(* CODESYS project SPT_Kinematics.library
   Placeholder: SPT Kinematics
   Title: SPT Kinematics
   Version: 3.3.5
   Company: Beckhoff Automation LLC

Project tree, tasks and I/O mapping:
  libraries: SPT Base Types, * (Beckhoff Automation LLC); SPT Components, * (Beckhoff Automation LLC); SPT Event Logger, * (Beckhoff Automation LLC); Tc2_MC2, * (Beckhoff Automation GmbH); Tc2_MC2_Camming, * (Beckhoff Automation GmbH); Tc2_NcKinematicTransformation, * (Beckhoff Automation GmbH); Tc2_Standard, * (Beckhoff Automation GmbH); Tc2_System, * (Beckhoff Automation GmbH); Tc3_EventLogger, * (Beckhoff Automation GmbH); Tc3_McCoordinatedMotion, * (Beckhoff Automation GmbH)
  DUTs/
    KinematicComponentAmp/
      Enumerations/
        data type E_InitializeState_KinematicAmp
      HMI/
        data type ST_KinematicComponentAmp_Command
        data type ST_KinematicComponentAmp_Config
        data type ST_KinematicComponentAmp_HMI
        data type ST_KinematicComponentAmp_Status
      data type ST_AmpPoint
      data type ST_AmpPointCircular
      data type ST_KinematicComponentAmp_CmGroupState
    KinematicComponentBase/
      Enumerations/
        data type E_InitializeState_KinematicComponent
        data type E_KinematicDOF
        data type E_KinematicEnableSeq
      HMI/
        data type ST_KinematicComponent_Command
        data type ST_KinematicComponent_Config
        data type ST_KinematicComponent_HMI
        data type ST_KinematicComponent_Status
        data type ST_KinematicJogCommand
      data type ST_BasePoint
      data type ST_KinematicMotionParameter
      data type ST_KinematicMotionParameterValues
      data type ST_KinematicPosition
    KinematicComponentCamming/
      Enumerations/
        data type E_InitializeState_KinematicCamming
      HMI/
        data type ST_KinematicComponentCam_Command
        data type ST_KinematicComponentCam_Config
        data type ST_KinematicComponentCam_HMI
        data type ST_KinematicComponentCam_Status
      data type ST_CamTableSlaveDynamics
    KinematicGroup/
      HMI/
        data type ST_KinematicGroup_Command
        data type ST_KinematicGroup_Config
        data type ST_KinematicGroup_HMI
        data type ST_KinematicGroup_Status
      data type E_ChangeParameterSeq
      data type E_InitializeState_KinematicGroup
      data type E_KinematicPositionCalculationSeq
    data type E_AcsJoint
    data type E_McsAxis
  FunctionBlocks/
    function block FB_ComponentKinematicBase [ST]: CreateEvents, HMICommunication, Monitoring, Reset, CyclicLogic, ActPosition, Enabled, InPosition, Moving, Disable, Enable, JogCartesianAxis, JogJoint, Override, Stop, TargetMotionParameter, BuildKinGroup, DissolveKinGroup, KinematicEnableSeq, McResetAllAxis, iAxisRef, Initialize
    function block FB_ComponentKinematicMotionAmp [ST]: CreateEvents, HMICommunication, Monitoring, Reset, CyclicLogic, Moving, Override, Stop, CmIdentAxis1, CmIdentAxis2, CmIdentAxis3, CmIdentAxis4, ConveyorRef, BuildCmGroup, ClearPath, CmGroupRef, CmState, DisableCmGroup, EnableCmGroup, SetCoordinateTransform, StartMovePath, TrackConveyorBelt, UngroupCmGroup, AddCircularMoveToPath, AddLinearMoveToPath, MoveToPointCartesian, ChangeOccurred, GetPoint, Points, SetPoint, Initialize
    function block FB_ComponentKinematicMotionCamming [ST]: CreateEvents, HMICommunication, Monitoring, Reset, CyclicLogic, Disable, Enable, Override, Stop, CamClearPath, CamIn, CamMasterZero, CammingActive, CamOut, CamStartMovePath, BuildKinGroup, DissolveKinGroup, ReadCamTableSlaveDynamicsACS, ReadCamTableSlaveDynamicsMCS, CamAddMotionPointByAxis, CamAddPointToPath, ChangeOccurred, GetPoint, Points, SetPoint, CamInOptionsACS, CamInOptionsMCS, CamMasterAcs, CamMasterMcs, CamTableSlaveDynamicsACS, CamTableSlaveDynamicsMCS, Initialize
    function block FB_KinematicAxisRef [ST]: ACS, AcsAxisCount, AcsPositionAbsolute, DegreesOfFreedomConfigured, MCS
    function block FB_KinematicCamming [ST]: CyclicLogic, CamClearPath, CamIn, CamMasterZero, CammingActive, CamOut, CamStartMovePath, CamAddMotionPointByAxis, CamAddPointToPath, CamTableAddStartPoint, Disable, Enable, ReadCamTableSlaveDynamics, Reset, SetOverride, Stop, CamAxisCount, CamAxisRef, CamInOptions, CamMaster, CamTableSlaveDynamics, Initialize
    function block FB_KinematicGroup [ST]: CreateEvents, HMICommunication, Monitoring, Reset, CyclicLogic, ActivateExtRotationRange, BuildKinGroup, DeactivateExtRotationRange, DissolveKinGroup, PresetRotationExtRotationRange, ResetKinGroup, SetKinematicParameter, KinematicStatus, KinMetaInfo, OidKinTrafo, OidKinTrafoTool, CalcKinPosition, ChangeKinematicParameter, KinematicAxisIds, Initialize
    function block FB_KinematicMotionAmpBase [ST]: CyclicLogic, BuildCmGroup, ClearPath, DisableCmGroup, EnableCmGroup, SetCoordinateTransform, StartMovePath, TrackConveyorBelt, UngroupCmGroup, CmIdentAxis1, CmIdentAxis2, CmIdentAxis3, CmIdentAxis4, ConveyorRef, CmGroupRef, CmState, AddCircularMoveToPath, AddLinearMoveToPath, MapStatus, Reset, SetOverride, Stop, CmAxisCount, CmAxisRef, Initialize
    function block FB_RingBuffer_AmpAmpPath [ST]: ClearPath, CurrentFB, GetNewFb, Path
  GVLs/
    global variables KINEMATIC_CONSTANTS
  Interfaces/
    interface I_Kinematic: Disable, Enable, JogCartesianAxis, JogJoint, Stop, ActPosition, Enabled, InPosition, Moving, Override, TargetMotionParameter
    interface I_KinematicAxisRef: ACS, AcsAxisCount, AcsPositionAbsolute, DegreesOfFreedomConfigured, MCS
    interface I_KinematicCamming: CamClearPath, CamIn, CamMasterZero, CamOut, CamStartMovePath, CammingActive
    interface I_KinematicCm: BuildCmGroup, ClearPath, DisableCmGroup, EnableCmGroup, SetCoordinateTransform, StartMovePath, TrackConveyorBelt, UngroupCmGroup, CmIdentAxis1, CmIdentAxis2, CmIdentAxis3, CmIdentAxis4, ConveyorRef, CmGroupRef, CmState
    interface I_KinematicGroup: ActivateExtRotationRange, BuildKinGroup, DeactivateExtRotationRange, DissolveKinGroup, PresetRotationExtRotationRange, ResetKinGroup, SetKinematicParameter, KinematicStatus, KinMetaInfo, OidKinTrafo, OidKinTrafoTool
  Project Information/
    function F_GetCompany [ST]
    function F_GetTitle [ST]
    function F_GetVersion [ST]
  Utilities/
    function F_ADSErrorCodeExt [ST]
  Version/
    global variables Global_Version
  00000000-0000-0000-0000-000000000000|LICENSE
  LICENSE
  global variables Parameter_Kinematic
*)

// DUTs/KinematicComponentAmp/Enumerations/E_InitializeState_KinematicAmp
{attribute 'qualified_only'}
{attribute 'strict'}
TYPE E_InitializeState_KinematicAmp : (
		eInitializeState_Start := 0,
		eInitializeState_CheckLinking,
		eInitializeState_Done,
		eInitializeState_Failed
	);
END_TYPE

// DUTs/KinematicComponentAmp/HMI/ST_KinematicComponentAmp_Command
TYPE ST_KinematicComponentAmp_Command :
	STRUCT
		BuildCmGroup	: BOOL;
		EnableCmGroup	: BOOL;
		PointSelect		: UDINT;
		MoveToPointCm	: BOOL;
		TeachPoint		: BOOL;
		DisableCmGroup	: BOOL;
		DissolveCmGroup : BOOL;
	END_STRUCT
END_TYPE

// DUTs/KinematicComponentAmp/HMI/ST_KinematicComponentAmp_Config
TYPE ST_KinematicComponentAmp_Config :
	STRUCT
		CustomOverride : BOOL := FALSE;
		CustomCommand  : DINT;
	END_STRUCT
END_TYPE

// DUTs/KinematicComponentAmp/HMI/ST_KinematicComponentAmp_HMI
TYPE ST_KinematicComponentAmp_HMI :
	STRUCT
		Config	: ST_KinematicComponentAmp_Config;
		Command : ST_KinematicComponentAmp_Command;
		Status	: ST_KinematicComponentAmp_Status;
	END_STRUCT
END_TYPE

// DUTs/KinematicComponentAmp/HMI/ST_KinematicComponentAmp_Status
TYPE ST_KinematicComponentAmp_Status :
	STRUCT
		CmState		  : ST_KinematicComponentAmp_CmGroupState;
		SelectedPoint : ST_AmpPoint;
	END_STRUCT
END_TYPE

// DUTs/KinematicComponentAmp/ST_AmpPoint
TYPE ST_AmpPoint EXTENDS ST_BasePoint :
	STRUCT
		CircularMove			 : ST_AmpPointCircular;
		Velocity				 : MC_LREAL			  := MC_INVALID;
		Acceleration			 : MC_LREAL			  := MC_DEFAULT;
		Deceleration			 : MC_LREAL			  := MC_DEFAULT;
		Jerk					 : MC_LREAL			  := MC_DEFAULT;
		BufferMode				 : MC_BUFFER_MODE	  := MC_BUFFER_MODE.mcAborting;
		TransitionMode			 : MC_TRANSITION_MODE := mcTransModeNone;
		TransitionParameter		 : ARRAY[1..2] OF LREAL;
		TransitionParameterCount : UDINT;
		InvokeId				 : UDINT;
	END_STRUCT
END_TYPE

// DUTs/KinematicComponentAmp/ST_AmpPointCircular
TYPE ST_AmpPointCircular :
	STRUCT
		IsCircularMove : BOOL;
		CircMode	   : MC_CIRC_MODE;
		AuxPoint	   : ARRAY[1..3] OF MC_LREAL;
		PathChoice	   : MC_CIRC_PATHCHOICE;
	END_STRUCT
END_TYPE

// DUTs/KinematicComponentAmp/ST_KinematicComponentAmp_CmGroupState
TYPE ST_KinematicComponentAmp_CmGroupState :
	STRUCT
		McToPlcCm					: CDT_MCTOPLC_GROUP_CM;
		GroupBuilt					: BOOL;
		GroupMoving					: BOOL;
		GroupHoming					: BOOL;
		GroupErrorStop				: BOOL;
		GroupNotReady				: BOOL;
		GroupStandby				: BOOL;
		GroupStopping				: BOOL;
		GroupDisabled				: BOOL;
		GroupTrackingInSync			: BOOL;
		GroupTrackingActive			: BOOL;
		GroupTrackingCommandAborted : BOOL;
		AllAxesStanding				: BOOL;
		ConstantVelocity			: BOOL;
		Accelerating				: BOOL;
		Decelerating				: BOOL;
		InPosition					: BOOL;
		Error						: BOOL;
		ErrorId						: UDINT;
	END_STRUCT
END_TYPE

// DUTs/KinematicComponentBase/Enumerations/E_InitializeState_KinematicComponent
{attribute 'qualified_only'}
{attribute 'strict'}
TYPE E_InitializeState_KinematicComponent : (
		eInitializeState_Start := 0,
		eInitializeState_CheckIft,
		eInitializeState_CheckAxisLinks,
		eInitializeState_SetAxisIds,
		eInitializeState_InitGroup,
		eInitializeState_Done
	);
END_TYPE

// DUTs/KinematicComponentBase/Enumerations/E_KinematicDOF
{attribute 'qualified_only'}
{attribute 'strict'}
TYPE E_KinematicDOF : (
		eKinematicDOF_2	  := 2, //
		eKinematicDOF_3	  := 3, //
		eKinematicDOF_4	  := 4, // 
		eKinematicDOF_5	  := 5, // 
		eKinematicDOF_6	  := 6, //
		eKinematicDOF_Max := 7	// 
	);
END_TYPE

// DUTs/KinematicComponentBase/Enumerations/E_KinematicEnableSeq
{attribute 'qualified_only'}
{attribute 'strict'}
TYPE E_KinematicEnableSeq : (
		eKinematicEnableSeq_Idle := 0,
		eKinematicEnableSeq_Start,
		eKinematicEnableSeq_ResetGroup,
		eKinematicEnableSeq_Enable,
		eKinematicEnableSeq_BuildGroup,
		eKinematicEnableSeq_Done
	);
END_TYPE

// DUTs/KinematicComponentBase/HMI/ST_KinematicComponent_Command
TYPE ST_KinematicComponent_Command :
	STRUCT
		Enable	: BOOL;
		Disable : BOOL;
		Stop	: BOOL;
		JogAxis : ARRAY[1..6] OF ST_KinematicJogCommand;
	END_STRUCT
END_TYPE

// DUTs/KinematicComponentBase/HMI/ST_KinematicComponent_Config
TYPE ST_KinematicComponent_Config :
	STRUCT
		KinematicType : E_KinematicDOF;
		AcsAxisCount  : UDINT;
	END_STRUCT
END_TYPE

// DUTs/KinematicComponentBase/HMI/ST_KinematicComponent_HMI
TYPE ST_KinematicComponent_HMI :
	STRUCT
		Config	: ST_KinematicComponent_Config;
		Command : ST_KinematicComponent_Command;
		Status	: ST_KinematicComponent_Status;
	END_STRUCT
END_TYPE

// DUTs/KinematicComponentBase/HMI/ST_KinematicComponent_Status
TYPE ST_KinematicComponent_Status :
	STRUCT
		Enabled		: BOOL;
		InPosition	: BOOL;
		Moving		: BOOL;
		ActPosition : ST_KinematicPosition;
	END_STRUCT
END_TYPE

// DUTs/KinematicComponentBase/HMI/ST_KinematicJogCommand
TYPE ST_KinematicJogCommand :
	STRUCT
		JogFast_Forward	 : BOOL;
		JogFast_Backward : BOOL;
		JogSlow_Forward	 : BOOL;
		JogSlow_Backward : BOOL;
	END_STRUCT
END_TYPE

// DUTs/KinematicComponentBase/ST_BasePoint
TYPE ST_BasePoint :
	STRUCT
		AcsPosition : ARRAY[1..KINEMATIC_CONSTANTS.DEGREES_OF_FREEDOM_MAX] OF LREAL;
		McsPosition : ARRAY[1..KINEMATIC_CONSTANTS.DEGREES_OF_FREEDOM_MAX] OF LREAL;
	END_STRUCT
END_TYPE

// DUTs/KinematicComponentBase/ST_KinematicMotionParameter
TYPE ST_KinematicMotionParameter :
	STRUCT
		Acs : ARRAY[1..KINEMATIC_CONSTANTS.DEGREES_OF_FREEDOM_MAX] OF ST_KinematicMotionParameterValues;
		Mcs : ARRAY[1..KINEMATIC_CONSTANTS.DEGREES_OF_FREEDOM_MAX] OF ST_KinematicMotionParameterValues;
	END_STRUCT
END_TYPE

// DUTs/KinematicComponentBase/ST_KinematicMotionParameterValues
TYPE ST_KinematicMotionParameterValues :
	STRUCT
		Position	 : LREAL;
		Acceleration : LREAL;
		Deceleration : LREAL;
		Jerk		 : LREAL;
	END_STRUCT
END_TYPE

// DUTs/KinematicComponentBase/ST_KinematicPosition
TYPE ST_KinematicPosition :
	STRUCT
		ACS : ARRAY[1..8] OF LREAL;
		MCS : ARRAY[1..8] OF LREAL;
	END_STRUCT
END_TYPE

// DUTs/KinematicComponentCamming/Enumerations/E_InitializeState_KinematicCamming
{attribute 'qualified_only'}
{attribute 'strict'}
TYPE E_InitializeState_KinematicCamming : (
		eInitializeState_Start := 0,
		eInitializeState_CheckLinking,
		eInitializeState_CheckRef,
		eInitializeState_Done,
		eInitializeState_Failed
	);
END_TYPE

// DUTs/KinematicComponentCamming/HMI/ST_KinematicComponentCam_Command
TYPE ST_KinematicComponentCam_Command :
	STRUCT
		CamAddPoint	   : BOOL;
		CamIn		   : BOOL;
		CamOut		   : BOOL;
		CamDeletePoint : BOOL;
		PointSelect	   : UDINT;
		MoveToPointCam : BOOL;
		TeachPoint	   : BOOL;
	END_STRUCT
END_TYPE

// DUTs/KinematicComponentCamming/HMI/ST_KinematicComponentCam_Config
TYPE ST_KinematicComponentCam_Config :
	STRUCT
		CustomOverride : BOOL := FALSE;
		CustomCommand  : DINT;
	END_STRUCT
END_TYPE

// DUTs/KinematicComponentCamming/HMI/ST_KinematicComponentCam_HMI
TYPE ST_KinematicComponentCam_HMI :
	STRUCT
		Config	: ST_KinematicComponentCam_Config;
		Command : ST_KinematicComponentCam_Command;
		Status	: ST_KinematicComponentCam_Status;
	END_STRUCT
END_TYPE

// DUTs/KinematicComponentCamming/HMI/ST_KinematicComponentCam_Status
TYPE ST_KinematicComponentCam_Status :
	STRUCT
		CammingActive : BOOL;
		SelectedPoint : ST_BasePoint;
	END_STRUCT
END_TYPE

// DUTs/KinematicComponentCamming/ST_CamTableSlaveDynamics
TYPE ST_CamTableSlaveDynamics :
	STRUCT
		SlavePosition	  : LREAL;
		SlaveVelocity	  : LREAL;
		SlaveAcceleration : LREAL;
	END_STRUCT
END_TYPE

// DUTs/KinematicGroup/HMI/ST_KinematicGroup_Command
TYPE ST_KinematicGroup_Command :
	STRUCT
		BuildGroup	  : BOOL;
		DissolveGroup : BOOL;
	END_STRUCT
END_TYPE

// DUTs/KinematicGroup/HMI/ST_KinematicGroup_Config
TYPE ST_KinematicGroup_Config :
	STRUCT
	END_STRUCT
END_TYPE

// DUTs/KinematicGroup/HMI/ST_KinematicGroup_HMI
TYPE ST_KinematicGroup_HMI :
	STRUCT
		Config	: ST_KinematicGroup_Config;
		Command : ST_KinematicGroup_Command;
		Status	: ST_KinematicGroup_Status;
	END_STRUCT
END_TYPE

// DUTs/KinematicGroup/HMI/ST_KinematicGroup_Status
TYPE ST_KinematicGroup_Status :
	STRUCT
		KinStatusReady : BOOL;
		KinStatus	   : E_KinStatus;
	END_STRUCT
END_TYPE

// DUTs/KinematicGroup/E_ChangeParameterSeq
{attribute 'qualified_only'}
{attribute 'strict'}
TYPE E_ChangeParameterSeq : (
		eChangeParameterSeq_Idle := 0,
		eChangeParameterSeq_Start,
		eChangeParameterSeq_Unlock,
		eChangeParameterSeq_Change,
		eChangeParameterSeq_ChangeDone,
		eChangeParameterSeq_Lock,
		eChangeParameterSeq_Error
	);
END_TYPE

// DUTs/KinematicGroup/E_InitializeState_KinematicGroup
{attribute 'qualified_only'}
{attribute 'strict'}
TYPE E_InitializeState_KinematicGroup : (
		eInitializeState_Start := 0,
		eInitializeState_CheckAxisIds,
		eInitializeState_CheckLinking,
		eInitializeState_CheckOid,
		eInitializeState_Done
	);
END_TYPE

// DUTs/KinematicGroup/E_KinematicPositionCalculationSeq
{attribute 'qualified_only'}
{attribute 'strict'}
TYPE E_KinematicPositionCalculationSeq : (
		eKinematicPositionCalculationSeq_Start := 0,
		eKinematicPositionCalculationSeq_Calc,
		eKinematicPositionCalculationSeq_Done
	);
END_TYPE

// DUTs/E_AcsJoint
{attribute 'qualified_only'}
TYPE E_AcsJoint : (
		Joint_1 := 1,
		Joint_2 := 2,
		Joint_3 := 3,
		Joint_4 := 4,
		Joint_5 := 5,
		Joint_6 := 6
	);
END_TYPE

// DUTs/E_McsAxis
{attribute 'qualified_only'}
TYPE E_McsAxis : (
		X	 := 1,
		Y	 := 2,
		Z	 := 3,
		Rot1 := 4, // C1, Rx,..
		Rot2 := 5, // C2, Ry,..
		Rot3 := 6  // C3, Rz,..
	);
END_TYPE

// GVLs/KINEMATIC_CONSTANTS
{attribute 'qualified_only'}
VAR_GLOBAL CONSTANT
	DEGREES_OF_FREEDOM_MAX : UINT := (TO_UINT(E_KinematicDOF.eKinematicDOF_Max) - 1);
END_VAR

// Version/Global_Version
{attribute 'TcGenerated'}
{attribute 'no-analysis'}
{attribute 'linkalways'}
// This function has been automatically generated from the project information.
VAR_GLOBAL CONSTANT
	{attribute 'const_non_replaced'}
	stLibVersion_SPT_Kinematics : ST_LibVersion := (iMajor := 3, iMinor := 3, iBuild := 5, iRevision := 0, nFlags := 1, sVersion := '3.3.5');
END_VAR

// Parameter_Kinematic
{attribute 'qualified_only'}
VAR_GLOBAL CONSTANT
	PathBufferSize				   : UDINT(4096..32768) := 4096;
	MaxPoints					   : UDINT(0..500)		:= 10;
	DefaultStopDeceleration		   : LREAL				:= 1000;  // mm/s^2 or deg/s^2
	DefaultStopDecelerationJerk	   : LREAL				:= 10000; // mm/s^3 or deg/s^3
	MaxCammingPositionsPerTable	   : UDINT(2..30)		:= 5;	  // Max Positions per move Command in Camming
	CamDefaultMoveVelocity		   : LREAL				:= 100;	  // mm/s or deg/s
	CamDefaultMoveAcceleration	   : LREAL				:= 1000;  // mm/s^2 or deg/s^2
	CamDefaultMoveDeceleration	   : LREAL				:= 1000;  // mm/s^2 or deg/s^2
	CamDefaultMoveJerk			   : LREAL				:= 10000; // mm/s^3 or deg/s^3		
	ExecuteCamPeriodically		   : BOOL				:= FALSE;
	CamMasterAbsolute			   : BOOL				:= TRUE;
	CamSlaveAbsolute			   : BOOL				:= TRUE;
	CammingFirstPointInTableByUser : BOOL				:= FALSE;
END_VAR

// FunctionBlocks/FB_ComponentKinematicBase
FUNCTION_BLOCK FB_ComponentKinematicBase EXTENDS FB_KinematicGroup IMPLEMENTS I_Kinematic
VAR
	// Kinematic Axis
	iAxis	 : I_KinematicAxisRef;
	_AxisAcs : REFERENCE TO ARRAY[1..KINEMATIC_CONSTANTS.DEGREES_OF_FREEDOM_MAX] OF AXIS_REF;
	_AxisMcs : REFERENCE TO ARRAY[1..KINEMATIC_CONSTANTS.DEGREES_OF_FREEDOM_MAX] OF AXIS_REF;

	// Internal Variables
	_KinematicComponentInit		: E_InitializeState_KinematicComponent;
	_KinematicEnableSeq			: E_KinematicEnableSeq := E_KinematicEnableSeq.eKinematicEnableSeq_Idle;
	_KinematicComponentBaseBusy : BOOL;
	_i							: UDINT;
	_ActPosition				: ST_KinematicPosition;
	_AcsSpeedOverride			: LREAL := 100.0;
	_McsSpeedOverride			: LREAL := 100.0;
	_McPowerAcsErrorActive		: BOOL;
	_McPowerMcsErrorActive		: BOOL;
	_TargetMotionParameter		: ST_KinematicMotionParameter;

	// MC Functions
	_McPowerACS : ARRAY[1..KINEMATIC_CONSTANTS.DEGREES_OF_FREEDOM_MAX] OF MC_POWER;
	_McPowerMCS : ARRAY[1..KINEMATIC_CONSTANTS.DEGREES_OF_FREEDOM_MAX] OF MC_POWER;
	_McJogACS	: ARRAY[1..KINEMATIC_CONSTANTS.DEGREES_OF_FREEDOM_MAX] OF MC_JOG;
	_McJogMCS	: ARRAY[1..KINEMATIC_CONSTANTS.DEGREES_OF_FREEDOM_MAX] OF MC_JOG;
	_McResetACS : ARRAY[1..KINEMATIC_CONSTANTS.DEGREES_OF_FREEDOM_MAX] OF MC_Reset;
	_McResetMCS : ARRAY[1..KINEMATIC_CONSTANTS.DEGREES_OF_FREEDOM_MAX] OF MC_Reset;
	_McHaltACS	: ARRAY[1..KINEMATIC_CONSTANTS.DEGREES_OF_FREEDOM_MAX] OF MC_Halt;
	_McHaltMCS	: ARRAY[1..KINEMATIC_CONSTANTS.DEGREES_OF_FREEDOM_MAX] OF MC_Halt;

	// HMI
	KinematicComponent_HMI : ST_KinematicComponent_HMI;

	// Alarms
	KinematicComponentBaseAlarms : ARRAY[1..KINEMATIC_COMPONENT_BASE_ALARM_COUNT] OF FB_TcAlarm;
END_VAR

VAR CONSTANT
	KINEMATIC_COMPONENT_BASE_ALARM_COUNT : UINT := 9;
END_VAR

//! @summary Initializes event function blocks using this components's name
{attribute 'call_after_online_change_slot' := '<slot>'}
METHOD PROTECTED CreateEvents

//! @description This method is called by <c>Initialize()</c> as required
F_CreateAllEventsInClass(Alarms		:= KinematicComponentBaseAlarms,
						 ClassSize	:= SIZEOF(TC_EVENTS.KinematicComponentBase),
						 pInitEvent := ADR(TC_EVENTS.KinematicComponentBase.InitReferenceEvent),
						 Prefix		:= Name);

SUPER^.CreateEvents();
END_METHOD

//! @summary Provides interlocks for HMI control and updates HMI status information for this component
METHOD PROTECTED HMICommunication

//! @description This method is called cyclically by <c>CyclicLogic()</c>
//Extend this method in extended FBs to communicate specific implementation data
SUPER^.HMICommunication();

// Kinematic HMI-Control
IF ComponentBase_HMI.Status.HMIControlAvailable THEN
	IF KinematicComponent_HMI.Command.Enable THEN
		THIS^.Enable();
		KinematicComponent_HMI.Command.Enable := FALSE;
	END_IF

	IF KinematicComponent_HMI.Command.Disable THEN
		THIS^.Disable();
		KinematicComponent_HMI.Command.Disable := FALSE;
	END_IF

	IF KinematicComponent_HMI.Command.Stop THEN
		Stop(0, 0);
		KinematicComponent_HMI.Command.Stop := FALSE;
	END_IF

	(*Jog*)
	FOR _i := 1 TO TO_UDINT(iAxis.DegreesOfFreedomConfigured) DO
		// Reset for Jogging-Function at HMI-control available
		THIS^.JogCartesianAxis(Axisx	:= _i,
							   Forward	:= FALSE,
							   Backward := FALSE,
							   JogMode	:= E_JogMode.MC_JOGMODE_STANDARD_SLOW);

		// Axis Jog Command
		IF SUPER^.KinematicStatus = E_KinStatus.KinStatus_Ready THEN // MCS-Axis active with Kinematic Model
			IF KinematicComponent_HMI.Command.JogAxis[_i].JogSlow_Forward THEN
				THIS^.JogCartesianAxis(Axisx	:= _i,
									   Forward	:= TRUE,
									   Backward := FALSE,
									   JogMode	:= E_JogMode.MC_JOGMODE_STANDARD_SLOW);
			ELSIF KinematicComponent_HMI.Command.JogAxis[_i].JogFast_Forward THEN
				THIS^.JogCartesianAxis(Axisx	:= _i,
									   Forward	:= TRUE,
									   Backward := FALSE,
									   JogMode	:= E_JogMode.MC_JOGMODE_STANDARD_FAST);
			ELSIF KinematicComponent_HMI.Command.JogAxis[_i].JogSlow_Backward THEN
				THIS^.JogCartesianAxis(Axisx	:= _i,
									   Forward	:= FALSE,
									   Backward := TRUE,
									   JogMode	:= E_JogMode.MC_JOGMODE_STANDARD_SLOW);
			ELSIF KinematicComponent_HMI.Command.JogAxis[_i].JogFast_Backward THEN
				THIS^.JogCartesianAxis(Axisx	:= _i,
									   Forward	:= FALSE,
									   Backward := TRUE,
									   JogMode	:= E_JogMode.MC_JOGMODE_STANDARD_FAST);
			END_IF
		END_IF
	END_FOR

	FOR _i := 1 TO TO_UDINT(iAxis.AcsAxisCount) DO
		// Reset for Jogging-Function at HMI-control available
		THIS^.JogJoint(Jointx	:= _i,
					   Forward	:= FALSE,
					   Backward := FALSE,
					   JogMode	:= E_JogMode.MC_JOGMODE_STANDARD_SLOW);

		// Axis Jog Command
		IF SUPER^.KinematicStatus = E_KinStatus.KinStatus_Empty THEN // ACS-Axis active
			IF KinematicComponent_HMI.Command.JogAxis[_i].JogSlow_Forward THEN
				THIS^.JogJoint(Jointx	:= _i,
							   Forward	:= TRUE,
							   Backward := FALSE,
							   JogMode	:= E_JogMode.MC_JOGMODE_STANDARD_SLOW);
			ELSIF KinematicComponent_HMI.Command.JogAxis[_i].JogFast_Forward THEN
				THIS^.JogJoint(Jointx	:= _i,
							   Forward	:= TRUE,
							   Backward := FALSE,
							   JogMode	:= E_JogMode.MC_JOGMODE_STANDARD_FAST);
			ELSIF KinematicComponent_HMI.Command.JogAxis[_i].JogSlow_Backward THEN
				THIS^.JogJoint(Jointx	:= _i,
							   Forward	:= FALSE,
							   Backward := TRUE,
							   JogMode	:= E_JogMode.MC_JOGMODE_STANDARD_SLOW);
			ELSIF KinematicComponent_HMI.Command.JogAxis[_i].JogFast_Backward THEN
				THIS^.JogJoint(Jointx	:= _i,
							   Forward	:= FALSE,
							   Backward := TRUE,
							   JogMode	:= E_JogMode.MC_JOGMODE_STANDARD_FAST);
			END_IF
		END_IF
	END_FOR
END_IF

// Status to HMI
KinematicComponent_HMI.Config.KinematicType := iAxis.DegreesOfFreedomConfigured;
KinematicComponent_HMI.Config.AcsAxisCount	:= iAxis.AcsAxisCount;
KinematicComponent_HMI.Status.Enabled		:= THIS^.Enabled;
KinematicComponent_HMI.Status.InPosition	:= THIS^.InPosition;
KinematicComponent_HMI.Status.Moving		:= THIS^.Moving;
KinematicComponent_HMI.Status.ActPosition	:= _ActPosition;
END_METHOD

//! Provides basic error detection and event handling for this component
METHOD PROTECTED Monitoring

(*! @descriptionThis method is called cyclically by <c>CyclicLogic()</c>*)
// Raise Error
SUPER^.Monitoring();
FOR _i := 1 TO TO_UDINT(iAxis.AcsAxisCount) DO
	IF _McPowerACS[_i].Error AND NOT KinematicComponentBaseAlarms[E_KinematicComponentBase.McPowerACS].bRaised THEN
		RaiseAlarmWithStrings(Alarm := KinematicComponentBaseAlarms[E_KinematicComponentBase.McPowerACS], F_ADSErrorCodeExt(_McPowerACS[_i].ErrorID), '');
		_McPowerAcsErrorActive := TRUE;
		EXIT;
	END_IF
END_FOR

// Raise Error
FOR _i := 1 TO TO_UDINT(iAxis.DegreesOfFreedomConfigured) DO
	IF _McPowerMCS[_i].Error AND NOT KinematicComponentBaseAlarms[E_KinematicComponentBase.McPowerMCS].bRaised THEN
		RaiseAlarmWithStrings(Alarm := KinematicComponentBaseAlarms[E_KinematicComponentBase.McPowerMCS], F_ADSErrorCodeExt(_McPowerMCS[_i].ErrorID), '');
		_McPowerMcsErrorActive := TRUE;
		EXIT;
	END_IF
END_FOR

// Raise Error
FOR _i := 1 TO TO_UDINT(iAxis.AcsAxisCount) DO
	IF _McJogACS[_i].Error AND NOT KinematicComponentBaseAlarms[E_KinematicComponentBase.McJogACS].bRaised THEN
		RaiseAlarmWithStrings(Alarm := KinematicComponentBaseAlarms[E_KinematicComponentBase.McJogACS], F_ADSErrorCodeExt(_McJogACS[_i].ErrorID), '');
	END_IF
END_FOR

// Raise Error
FOR _i := 1 TO TO_UDINT(iAxis.DegreesOfFreedomConfigured) DO
	IF _McJogMCS[_i].Error AND NOT KinematicComponentBaseAlarms[E_KinematicComponentBase.McJogMcs].bRaised THEN
		RaiseAlarmWithStrings(Alarm := KinematicComponentBaseAlarms[E_KinematicComponentBase.McJogMCS], F_ADSErrorCodeExt(_McJogMCS[_i].ErrorID), '');
		EXIT;
	END_IF
END_FOR

// Raise Error
FOR _i := 1 TO TO_UDINT(iAxis.AcsAxisCount) DO
	IF _McResetACS[_i].Error AND NOT KinematicComponentBaseAlarms[E_KinematicComponentBase.McResetACS].bRaised THEN
		RaiseAlarmWithStrings(Alarm := KinematicComponentBaseAlarms[E_KinematicComponentBase.McResetACS], F_ADSErrorCodeExt(_McResetACS[_i].ErrorID), '');
	END_IF
END_FOR

// Raise Error
FOR _i := 1 TO TO_UDINT(iAxis.DegreesOfFreedomConfigured) DO
	IF _McResetMCS[_i].Error AND NOT KinematicComponentBaseAlarms[E_KinematicComponentBase.McResetMcs].bRaised THEN
		RaiseAlarmWithStrings(Alarm := KinematicComponentBaseAlarms[E_KinematicComponentBase.McResetMCS], F_ADSErrorCodeExt(_McResetMCS[_i].ErrorID), '');
		EXIT;
	END_IF
END_FOR

// Raise Error
FOR _i := 1 TO TO_UDINT(iAxis.AcsAxisCount) DO
	IF _McHaltACS[_i].Error AND NOT KinematicComponentBaseAlarms[E_KinematicComponentBase.McHaltACS].bRaised THEN
		RaiseAlarmWithStrings(Alarm := KinematicComponentBaseAlarms[E_KinematicComponentBase.McHaltACS], F_ADSErrorCodeExt(_McHaltACS[_i].ErrorID), '');
	END_IF
END_FOR

// Raise Error
FOR _i := 1 TO TO_UDINT(iAxis.DegreesOfFreedomConfigured) DO
	IF _McHaltMCS[_i].Error AND NOT KinematicComponentBaseAlarms[E_KinematicComponentBase.McHaltMcs].bRaised THEN
		RaiseAlarmWithStrings(Alarm := KinematicComponentBaseAlarms[E_KinematicComponentBase.McHaltMCS], F_ADSErrorCodeExt(_McHaltMCS[_i].ErrorID), '');
		EXIT;
	END_IF
END_FOR

_CurrentAlarmSeverity := F_GetMaxSeverityRaised(Alarms := KinematicComponentBaseAlarms, CurrentSeverity := _CurrentAlarmSeverity);
END_METHOD

//! @summary Clears error flags and error IDs for this component
METHOD PUBLIC Reset : BOOL
FOR _i := 1 TO TO_UDINT(iAxis.DegreesOfFreedomConfigured) DO
	_McJogMcs[_i].JogForward   := FALSE;
	_McJogMcs[_i].JogBackwards := FALSE;
END_FOR

FOR _i := 1 TO TO_UDINT(iAxis.AcsAxisCount) DO
	_McJogAcs[_i].JogForward   := FALSE;
	_McJogAcs[_i].JogBackwards := FALSE;
END_FOR

// Remove Enable Singal at fatal Kinematic Error - trigger startup sequence following
IF _McPowerAcsErrorActive OR _McPowerMcsErrorActive THEN
	FOR _i := 1 TO TO_UDINT(iAxis.DegreesOfFreedomConfigured) DO
		_McPowerMcs[_i].Enable := FALSE;
	END_FOR

	FOR _i := 1 TO TO_UDINT(iAxis.AcsAxisCount) DO
		_McPowerAcs[_i].Enable := FALSE;
	END_FOR

	SUPER^.DissolveKinGroup(); // Dissolve Group after MC-Power error - startup from Joint mode in case of singularity
END_IF

IF THIS^.Error THEN
	// Reset Kinematic Axis ACS and MCS when error active
	THIS^.McResetAllAxis();
	_McPowerAcsErrorActive := FALSE;
	_McPowerMcsErrorActive := FALSE;
	F_ClearAllEventsInClass(KinematicComponentBaseAlarms);
END_IF

Reset := SUPER^.Reset();
END_METHOD

//! @summary This method serves as the entry point for all underlying FB logic
METHOD PUBLIC CyclicLogic
IF NOT _InitComplete THEN
	_InitComplete := Initialize();
	RETURN;
END_IF

// Call Kinematic FBs
FOR _i := 1 TO TO_UDINT(iAxis.AcsAxisCount) DO
	// Read Current Status
	iAxis.ACS[_i].ReadStatus();
	IF iAxis.AcsPositionAbsolute THEN
		_ActPosition.ACS[_i] := iAxis.ACS[_i].NcToPlc.ActPos;
	ELSE
		_ActPosition.ACS[_i] := iAxis.ACS[_i].NcToPlc.ModuloActPos; // ACS Joints are always rotational Modulo Drives 0..360 deg
	END_IF

	// Set Reference
	_AxisAcs REF= iAxis.ACS;
	{Region - MC_Power}
	_McPowerACS[_i](Axis			:= _AxisAcs[_i],
					Enable_Positive := TRUE,
					Enable_Negative := TRUE,
					Override		:= _AcsSpeedOverride);

	IF _McPowerACS[_i].Error THEN
		_Error	 := TRUE;
		_ErrorID := _McPowerACS[_i].ErrorID;
	END_IF

	{endregion}
	{Region - MC_Jog}
	_McJogACS[_i](Axis := _AxisAcs[_i]);
	IF _McJogACS[_i].Error THEN
		_Error	 := TRUE;
		_ErrorID := _McJogACS[_i].ErrorID;
	END_IF

	{endregion}
	{Region - MC_Reset}
	_McResetACS[_i](Axis := _AxisAcs[_i]);
	IF _McResetACS[_i].Error THEN
		_Error	 := TRUE;
		_ErrorID := _McResetACS[_i].ErrorID;
	END_IF

	_McResetACS[_i].Execute := FALSE;
	{endregion}
	{Region - MC_Halt}
	_McHaltACS[_i](Axis := _AxisAcs[_i]);
	IF _McHaltACS[_i].Error THEN
		_Error	 := TRUE;
		_ErrorID := _McHaltACS[_i].ErrorID;
	END_IF

	_McHaltACS[_i].Execute := FALSE;
	{endregion}
END_FOR

// Call Kinematic FBs
FOR _i := 1 TO TO_UDINT(iAxis.DegreesOfFreedomConfigured) DO
	// Read Current Status
	iAxis.MCS[_i].ReadStatus();

	// Set Reference
	_AxisMcs REF= iAxis.MCS;
	{Region - MC_Power}
	_McPowerMCS[_i](Axis			:= _AxisMcs[_i],
					Enable_Positive := TRUE,
					Enable_Negative := TRUE,
					Override		:= _McsSpeedOverride);

	IF _McPowerMCS[_i].Error THEN
		_Error	 := TRUE;
		_ErrorID := _McPowerMCS[_i].ErrorID;
	END_IF

	{endregion}
	{Region - MC_Jog}
	_McJogMCS[_i](Axis := _AxisMcs[_i]);
	IF _McJogMCS[_i].Error THEN
		_Error	 := TRUE;
		_ErrorID := _McJogMCS[_i].ErrorID;
	END_IF

	{endregion}
	{Region - MC_Reset}
	_McResetMCS[_i](Axis := _AxisMcs[_i]);
	IF _McResetMCS[_i].Error THEN
		_Error	 := TRUE;
		_ErrorID := _McResetMCS[_i].ErrorID;
	END_IF

	_McResetMCS[_i].Execute := FALSE;
	{endregion}
	{Region - MC_Halt}
	_McHaltMCS[_i](Axis := _AxisMcs[_i]);
	IF _McHaltMCS[_i].Error THEN
		_Error	 := TRUE;
		_ErrorID := _McHaltMCS[_i].ErrorID;
	END_IF

	_McHaltMCS[_i].Execute := FALSE;
	{endregion}
END_FOR

(* Startup Sequence for Kinematic in Cartesian Mode *)
KinematicEnableSeq();

(* Calculate MCS Position independent of built group *)
IF SUPER^.KinematicStatus = E_KinStatus.KinStatus_Ready THEN
	FOR _i := 1 TO TO_UDINT(iAxis.DegreesOfFreedomConfigured) DO
		IF _i <= E_McsAxis.Z THEN
			_ActPosition.MCS[_i] := iAxis.MCS[_i].NcToPlc.ActPos; // Real-Time Data from NC in Cartesian Mode
		ELSE
			_ActPosition.MCS[_i] := iAxis.MCS[_i].NcToPlc.ModuloActPos; // Real-Time Data from NC in Cartesian Mode, rotational Joints
		END_IF
	END_FOR
ELSE
	SUPER^.CalcKinPosition(ACS := _ActPosition.ACS, MCS => _ActPosition.MCS); // Calculate Posiiton 4x per s in Joint Mode
END_IF

(* Create Busy signal *)
THIS^._KinematicComponentBaseBusy := SUPER^._KinematicGroupBusy OR _KinematicEnableSeq <> E_KinematicEnableSeq.eKinematicEnableSeq_Idle;
FOR _i := 1 TO TO_UDINT(iAxis.DegreesOfFreedomConfigured) DO
	IF _McJogMCS[_i].Busy OR _McHaltMCS[_i].Busy THEN
		THIS^._KinematicComponentBaseBusy := TRUE;
		EXIT;
	END_IF
END_FOR

FOR _i := 1 TO TO_UDINT(iAxis.AcsAxisCount) DO
	IF _McJogACS[_i].Busy OR _McHaltACS[_i].Busy THEN
		THIS^._KinematicComponentBaseBusy := TRUE;
		EXIT;
	END_IF
END_FOR

SUPER^.CyclicLogic();
END_METHOD

{attribute 'monitoring' := 'variable'}
PROPERTY ActPosition : ST_KinematicPosition
GET
ActPosition := _ActPosition;
END_GET
END_PROPERTY

{attribute 'monitoring' := 'variable'}
PROPERTY PUBLIC Enabled : BOOL
GET
Enabled := FALSE;
FOR _i := 1 TO TO_UDINT(iAxis.DegreesOfFreedomConfigured) DO
	IF NOT _McPowerMCS[_i].Status THEN
		RETURN;
	END_IF
END_FOR

FOR _i := 1 TO TO_UDINT(iAxis.AcsAxisCount) DO
	IF NOT _McPowerACS[_i].Status THEN
		RETURN;
	END_IF
END_FOR

Enabled := TRUE;
END_GET
END_PROPERTY

{attribute 'monitoring' := 'variable'}
PROPERTY PUBLIC InPosition : BOOL
GET
InPosition := FALSE;
FOR _i := 1 TO TO_UDINT(iAxis.DegreesOfFreedomConfigured) DO
	IF NOT iAxis.MCS[_i].Status.InTargetPosition THEN
		RETURN;
	END_IF
END_FOR

FOR _i := 1 TO TO_UDINT(iAxis.AcsAxisCount) DO
	IF NOT iAxis.ACS[_i].Status.InTargetPosition THEN
		RETURN;
	END_IF
END_FOR

InPosition := TRUE;
END_GET
END_PROPERTY

{attribute 'monitoring' := 'variable'}
PROPERTY PUBLIC Moving : BOOL
GET
Moving := FALSE;
FOR _i := 1 TO TO_UDINT(iAxis.DegreesOfFreedomConfigured) DO
	IF NOT (iAxis.MCS[_i].NcToPlc.StateDWord.2) THEN // StatusDWord Bit 2 = Axis is logically stationary ("Axis not moving")

		// .Status.Moving is not valid if Kinematic reaches end of workspace fault
		Moving := TRUE;
	END_IF
END_FOR

FOR _i := 1 TO TO_UDINT(iAxis.AcsAxisCount) DO
	IF NOT (iAxis.ACS[_i].NcToPlc.StateDWord.2) THEN // StatusDWord Bit 2 = Axis is logically stationary ("Axis not moving")

		// .Status.Moving is not valid if Kinematic reaches end of workspace fault
		Moving := TRUE;
	END_IF
END_FOR
END_GET
END_PROPERTY

METHOD PUBLIC Disable : BOOL
Disable				:= FALSE;
_KinematicEnableSeq := E_KinematicEnableSeq.eKinematicEnableSeq_Idle;
FOR _i := 1 TO TO_UDINT(iAxis.DegreesOfFreedomConfigured) DO
	_McPowerMCS[_i].Enable := FALSE;
END_FOR

FOR _i := 1 TO TO_UDINT(iAxis.AcsAxisCount) DO
	_McPowerACS[_i].Enable := FALSE;
END_FOR

Disable := TRUE;
END_METHOD

METHOD PUBLIC Enable : BOOL
Enable := FALSE;
IF SUPER^.KinematicStatus = E_KinStatus.KinStatus_Empty THEN
	FOR _i := 1 TO TO_UDINT(iAxis.DegreesOfFreedomConfigured) DO
		_McPowerMCS[_i].Enable := TRUE;
	END_FOR

	FOR _i := 1 TO TO_UDINT(iAxis.AcsAxisCount) DO
		_McPowerACS[_i].Enable := TRUE;
	END_FOR
ELSE
	_KinematicEnableSeq := E_KinematicEnableSeq.eKinematicEnableSeq_Start;
END_IF

Enable := TRUE;
END_METHOD

METHOD JogCartesianAxis : BOOL
VAR_INPUT
	Axisx	 : UDINT(1..KINEMATIC_CONSTANTS.DEGREES_OF_FREEDOM_MAX);
	Forward	 : BOOL;
	Backward : BOOL;
	JogMode	 : E_JogMode;
END_VAR
JogCartesianAxis := FALSE;
IF Axisx > TO_UDINT(iAxis.DegreesOfFreedomConfigured) THEN
	TRACE('Jog Cartesian Axis - Selected Axis greater than configured Kinematic');
	RETURN;
END_IF

IF Forward OR Backward THEN
	IF SUPER^.KinematicStatus <> E_KinStatus.KinStatus_Ready THEN
		TRACE('Jog Cartesian Axis - not possible Kinematic not in Cartesian mode (Ready-state)!');
		RETURN;
	END_IF

	IF JogMode <> E_JogMode.MC_JOGMODE_STANDARD_FAST AND JogMode <> E_JogMode.MC_JOGMODE_STANDARD_SLOW THEN
		TRACE('Jog Cartesian Axis - Not supported Jog-Mode selected!');
		RETURN;
	END_IF
END_IF

_McJogMcs[Axisx].JogForward	  := Forward;
_McJogMcs[Axisx].JogBackwards := Backward;
_McJogMcs[Axisx].Mode		  := JogMode;
JogCartesianAxis			  := TRUE;
END_METHOD

METHOD JogJoint : BOOL
VAR_INPUT
	Jointx	 : UDINT(1..KINEMATIC_CONSTANTS.DEGREES_OF_FREEDOM_MAX);
	Forward	 : BOOL;
	Backward : BOOL;
	JogMode	 : E_JogMode;
END_VAR
JogJoint := FALSE;
IF Jointx > TO_UDINT(iAxis.AcsAxisCount) THEN
	TRACE('Jog Joint - Selected Joint greater than configured Kinematic!');
	RETURN;
END_IF

IF Forward OR Backward THEN
	IF SUPER^.KinematicStatus <> E_KinStatus.KinStatus_Empty THEN
		TRACE('Jog Joint - not possible Kinematic not in Joint mode (Empty-state)!');
		RETURN;
	END_IF

	IF JogMode <> E_JogMode.MC_JOGMODE_STANDARD_FAST AND JogMode <> E_JogMode.MC_JOGMODE_STANDARD_SLOW THEN
		TRACE('Jog Joint - Not supported Jog-Mode selected!');
		RETURN;
	END_IF
END_IF

_McJogACS[Jointx].JogForward   := Forward;
_McJogACS[Jointx].JogBackwards := Backward;
_McJogACS[Jointx].Mode		   := JogMode;
JogJoint					   := TRUE;
END_METHOD

{attribute 'monitoring' := 'variable'}
PROPERTY PUBLIC Override : LREAL
SET
IF _KinStatus = E_Kinstatus.KinStatus_Ready THEN
	_AcsSpeedOverride := 100.0;
	_McsSpeedOverride := Override;
ELSE
	_AcsSpeedOverride := Override;
	_McsSpeedOverride := 100.0;
END_IF
END_SET
END_PROPERTY

METHOD PUBLIC Stop : BOOL
VAR_INPUT
	(*In Kinematic Base FB deceleration Input and Jerk input for Stop() are not used. 
	Intention is that for each of the possible 6 Axis a different Dcc and Dcc-Jerk might be possible.
	If the Inputs are needed, the function can be overloaded and programmed as desired.*)
	Deceleration : LREAL;
	Jerk		 : LREAL;
END_VAR
IF _KinStatus = E_KinStatus.KinStatus_Ready THEN
	FOR _i := 1 TO TO_UDINT(iAxis.DegreesOfFreedomConfigured) DO
		_McHaltMcs[_i].Deceleration := _TargetMotionParameter.Mcs[_i].Deceleration;
		_McHaltMcs[_i].Jerk			:= _TargetMotionParameter.Mcs[_i].Jerk;
		_McHaltMcs[_i].Execute		:= TRUE;
	END_FOR
ELSE
	FOR _i := 1 TO TO_UDINT(iAxis.AcsAxisCount) DO
		_McHaltAcs[_i].Deceleration := _TargetMotionParameter.Acs[_i].Deceleration;
		_McHaltAcs[_i].Jerk			:= _TargetMotionParameter.Acs[_i].Jerk;
		_McHaltAcs[_i].Execute		:= TRUE;
	END_FOR
END_IF

Stop := TRUE;
END_METHOD

{attribute 'monitoring' := 'variable'}
PROPERTY TargetMotionParameter : REFERENCE TO ST_KinematicMotionParameter
GET
TargetMotionParameter REF= _TargetMotionParameter;
END_GET
END_PROPERTY

METHOD PUBLIC BuildKinGroup : BOOL
IF NOT THIS^.Enabled THEN
	TRACE('Build Kinematic Group not possible - ACS Axis System not enabled!');
	RETURN;
END_IF

IF _Busy THEN
	RETURN;
END_IF

BuildKinGroup := SUPER^.BuildKinGroup();
END_METHOD

METHOD PUBLIC DissolveKinGroup : BOOL
DissolveKinGroup := SUPER^.DissolveKinGroup();
END_METHOD

METHOD PROTECTED KinematicEnableSeq : BOOL
CASE _KinematicEnableSeq OF
	E_KinematicEnableSeq.eKinematicEnableSeq_Idle:
		; // Start executed from Methode Enable()
	E_KinematicEnableSeq.eKinematicEnableSeq_Start:
		IF SUPER^.KinematicStatus = E_KinStatus.KinStatus_Error THEN
			_KinematicEnableSeq := E_KinematicEnableSeq.eKinematicEnableSeq_ResetGroup;
		ELSE
			_KinematicEnableSeq := E_KinematicEnableSeq.eKinematicEnableSeq_Enable;
		END_IF

	E_KinematicEnableSeq.eKinematicEnableSeq_ResetGroup:
		THIS^.McResetAllAxis();
		IF SUPER^.KinematicStatus = E_KinStatus.KinStatus_Unknown THEN
			_KinematicEnableSeq := E_KinematicEnableSeq.eKinematicEnableSeq_Enable;
		END_IF

	E_KinematicEnableSeq.eKinematicEnableSeq_Enable:
		FOR _i := 1 TO TO_UDINT(iAxis.AcsAxisCount) DO
			_McPowerACS[_i].Enable := TRUE; // Enable ACS to Start Kinematic
		END_FOR

		IF SUPER^.KinematicStatus = E_KinStatus.KinStatus_StartPending THEN
			_KinematicEnableSeq := E_KinematicEnableSeq.eKinematicEnableSeq_BuildGroup;
		END_IF

		IF SUPER^.KinematicStatus = E_KinStatus.KinStatus_Ready THEN
			_KinematicEnableSeq := E_KinematicEnableSeq.eKinematicEnableSeq_Done;
		END_IF

	E_KinematicEnableSeq.eKinematicEnableSeq_BuildGroup:
		SUPER^.BuildKinGroup();
		IF SUPER^.KinematicStatus = E_KinStatus.KinStatus_Ready THEN
			_KinematicEnableSeq := E_KinematicEnableSeq.eKinematicEnableSeq_Done;
		END_IF

	E_KinematicEnableSeq.eKinematicEnableSeq_Done:
		FOR _i := 1 TO TO_UDINT(iAxis.DegreesOfFreedomConfigured) DO
			_McPowerMCS[_i].Enable := TRUE; // Enable MCS to Start Kinematic
		END_FOR

		_KinematicEnableSeq := E_KinematicEnableSeq.eKinematicEnableSeq_Idle;
END_CASE
END_METHOD

METHOD PROTECTED McResetAllAxis : BOOL
VAR_INPUT
END_VAR
FOR _i := 1 TO TO_UDINT(iAxis.DegreesOfFreedomConfigured) DO
	_McResetMcs[_i].Execute := TRUE;
END_FOR

FOR _i := 1 TO TO_UDINT(iAxis.AcsAxisCount) DO
	_McResetAcs[_i].Execute := TRUE;
END_FOR

McResetAllAxis := TRUE;
END_METHOD

PROPERTY iAxisRef : I_KinematicAxisRef
SET
iAxis := iAxisRef;
END_SET
END_PROPERTY

//! @summary Basic component initialization logic
METHOD PROTECTED Initialize : BOOL;
CASE _KinematicComponentInit OF
	E_InitializeState_KinematicComponent.eInitializeState_Start:
		_KinematicEnableSeq		:= E_KinematicEnableSeq.eKinematicEnableSeq_Idle;
		_KinematicComponentInit := E_InitializeState_KinematicComponent.eInitializeState_CheckIft;

	E_InitializeState_KinematicComponent.eInitializeState_CheckIft:
		IF iAxis = 0 THEN
			Trace(CONCAT('Programming Error init failed with Interface to AxisRef missing - ', Name));
			_Busy  := FALSE;
			_Error := TRUE;
		ELSE
			_KinematicComponentInit := E_InitializeState_KinematicComponent.eInitializeState_CheckAxisLinks;
		END_IF

	E_InitializeState_KinematicComponent.eInitializeState_CheckAxisLinks:
		_KinematicComponentInit := E_InitializeState_KinematicComponent.eInitializeState_SetAxisIds;
		FOR _i := 1 TO TO_UDINT(iAxis.DegreesOfFreedomConfigured) DO
			IF F_GetMappingStatus(ADR(iAxis.MCS[_i].NcToPlc), SIZEOF(iAxis.MCS[_i].NcToPlc)) <> EPlcMappingStatus.MS_Mapped THEN
				Trace(CONCAT('Programming Error init failed with Axis Links missing - ', Name));
				_Busy  := FALSE;
				_Error := TRUE;
				EXIT;
			END_IF
		END_FOR

		FOR _i := 1 TO TO_UDINT(iAxis.AcsAxisCount) DO
			IF F_GetMappingStatus(ADR(iAxis.ACS[_i].NcToPlc), SIZEOF(iAxis.ACS[_i].NcToPlc)) <> EPlcMappingStatus.MS_Mapped THEN
				Trace(CONCAT('Programming Error init failed with Axis Links missing - ', Name));
				_Busy  := FALSE;
				_Error := TRUE;
				EXIT;
			END_IF
		END_FOR

	E_InitializeState_KinematicComponent.eInitializeState_SetAxisIds:
		FOR _i := 1 TO TO_UDINT(iAxis.DegreesOfFreedomConfigured) DO
			SUPER^.KinematicAxisIds.nAxisIdsMcs[_i] := iAxis.MCS[_i].NcToPlc.AxisId;
			IF SUPER^.KinematicAxisIds.nAxisIdsMcs[_i] = 0 THEN
				TRACE(CONCAT('Axis-Id missing MCS - ', Name));
				RETURN;
			END_IF
		END_FOR

		FOR _i := 1 TO TO_UDINT(iAxis.AcsAxisCount) DO
			SUPER^.KinematicAxisIds.nAxisIdsAcs[_i] := iAxis.ACS[_i].NcToPlc.AxisId;
			IF SUPER^.KinematicAxisIds.nAxisIdsAcs[_i] = 0 THEN
				TRACE(CONCAT('Axis-Id missing ACS - ', Name));
				RETURN;
			END_IF
		END_FOR

		_KinematicComponentInit := E_InitializeState_KinematicComponent.eInitializeState_InitGroup;

	E_InitializeState_KinematicComponent.eInitializeState_InitGroup:
		IF SUPER^.Initialize() THEN
			_KinematicComponentInit := E_InitializeState_KinematicComponent.eInitializeState_Done;
		END_IF

	E_InitializeState_KinematicComponent.eInitializeState_Done:
		_Busy	   := FALSE;
		Initialize := TRUE;
END_CASE
END_METHOD

END_FUNCTION_BLOCK

// FunctionBlocks/FB_KinematicGroup
FUNCTION_BLOCK FB_KinematicGroup EXTENDS FB_ComponentBase IMPLEMENTS I_KinematicGroup
VAR
	// Kinematic Channel
	KinematicChannelNcToPlc AT %I* : NCTOPLC_NCICHANNEL_REF; // Input Connection to Kinematic Channel
	KinematicChannelPlcToNc AT %Q* : PLCTONC_NCICHANNEL_REF; // Output Connection to Kinematic Channel

	// Internal Variables
	_KinematicGroupInit				 : E_InitializeState_KinematicGroup;
	_KinematicPositionCalculationSeq : E_KinematicPositionCalculationSeq := E_KinematicPositionCalculationSeq.eKinematicPositionCalculationSeq_Start;
	_KinAxisIds						 : ST_KinAxes; // ID-List of depending Axis for Kinematic 
	_KinConfigGroup					 : FB_KinConfigGroup;
	_KinResetGroup					 : FB_KinResetGroup;
	_KinStatus						 : E_KinStatus;
	_KinematicGroupBusy				 : BOOL; // Base object is busy
	{attribute 'TcInitSymbol'}
	_OidKinTrafo : OTCID;
	{attribute 'TcInitSymbol'}
	_OidKinTrafoTool		  : OTCID;
	_KinMetaInfoIn			  : U_KinMetaInfo;
	_KinMetaInfoOut			  : U_KinMetaInfo;
	_KinCalcTrafo			  : FB_KinCalcTrafo;
	_ChangeParameterSeq		  : E_ChangeParameterSeq := E_ChangeParameterSeq.eChangeParameterSeq_Idle;
	_KinUnlockTrafoParam	  : FB_KinUnlockTrafoParam;
	_KinLockTrafoParam		  : FB_KinLockTrafoParam;
	_AdsWrite				  : ADSWRITE;
	_KinPTCID				  : PTCID;
	_KinExtendedRotationRange : FB_KinExtendedRotationRange;
	_KinPresetRotation		  : FB_KinPresetRotation;
	_Rotation				  : ARRAY[1..3] OF LREAL; // Relates to 3 rotations availabe

	// Timer
	_KinCalcMcsPosition : TON;

	// HMI
	KinematicGroup_HMI : ST_KinematicGroup_HMI;

	// Alarms
	KinematicGroupAlarms : ARRAY[1..KINEMATIC_GROUP_ALARM_COUNT] OF FB_TcAlarm;
END_VAR

VAR CONSTANT
	KINEMATIC_GROUP_ALARM_COUNT : UINT := 9;
END_VAR

//! @summary Initializes event function blocks using this components's name
{attribute 'call_after_online_change_slot' := '<slot>'}
METHOD PROTECTED CreateEvents

//! @description This method is called by <c>Initialize()</c> as required
F_CreateAllEventsInClass(Alarms		:= KinematicGroupAlarms,
						 ClassSize	:= SIZEOF(TC_EVENTS.KinematicGroup),
						 pInitEvent := ADR(TC_EVENTS.KinematicGroup.InitReferenceEvent),
						 Prefix		:= Name);

SUPER^.CreateEvents();
END_METHOD

//! @summary Provides interlocks for HMI control and updates HMI status information for this component
METHOD PROTECTED HMICommunication

//! @description This method is called cyclically by <c>CyclicLogic()</c>
//Extend this method in extended FBs to communicate specific implementation data
SUPER^.HMICommunication();

// Kinematic HMI-Control
IF ComponentBase_HMI.Status.HMIControlAvailable THEN
	IF NOT _Busy AND KinematicGroup_HMI.Command.DissolveGroup THEN
		THIS^.DissolveKinGroup();
		KinematicGroup_HMI.Command.DissolveGroup := FALSE;
	END_IF

	IF NOT _Busy AND KinematicGroup_HMI.Command.BuildGroup THEN
		THIS^.BuildKinGroup();
		KinematicGroup_HMI.Command.BuildGroup := FALSE;
	END_IF
END_IF

// Status to HMI
KinematicGroup_HMI.Status.KinStatus		 := _KinStatus;
KinematicGroup_HMI.Status.KinStatusReady := _KinStatus = E_KinStatus.KinStatus_Ready;
END_METHOD

//! Provides basic error detection and event handling for this component
METHOD PROTECTED Monitoring

(*! @descriptionThis method is called cyclically by <c>CyclicLogic()</c>*)
SUPER^.Monitoring();
IF _KinConfigGroup.bError AND NOT KinematicGroupAlarms[E_KinematicGroup.KinConfigGroup].bRaised THEN
	RaiseAlarmWithStrings(Alarm := KinematicGroupAlarms[E_KinematicGroup.KinConfigGroup], F_ADSErrorCodeExt(_KinConfigGroup.nErrorId), '');
END_IF

IF _KinUnlockTrafoParam.bError AND NOT KinematicGroupAlarms[E_KinematicGroup.UnlockTrafoParam].bRaised THEN
	RaiseAlarmWithStrings(Alarm := KinematicGroupAlarms[E_KinematicGroup.UnlockTrafoParam], F_ADSErrorCodeExt(_KinUnlockTrafoParam.nErrorId), '');
END_IF

IF _KinLockTrafoParam.bError AND NOT KinematicGroupAlarms[E_KinematicGroup.LockTrafoParam].bRaised THEN
	RaiseAlarmWithStrings(Alarm := KinematicGroupAlarms[E_KinematicGroup.LockTrafoParam], F_ADSErrorCodeExt(_KinLockTrafoParam.nErrorId), '');
END_IF

IF _KinExtendedRotationRange.bError AND NOT KinematicGroupAlarms[E_KinematicGroup.ActivateExtRotation].bRaised THEN
	RaiseAlarmWithStrings(Alarm := KinematicGroupAlarms[E_KinematicGroup.ActivateExtRotation], F_ADSErrorCodeExt(_KinExtendedRotationRange.nErrorId), '');
END_IF

IF _KinPresetRotation.bError AND NOT KinematicGroupAlarms[E_KinematicGroup.PresetExtRotation].bRaised THEN
	RaiseAlarmWithStrings(Alarm := KinematicGroupAlarms[E_KinematicGroup.PresetExtRotation], F_ADSErrorCodeExt(_KinPresetRotation.nErrorId), '');
END_IF

_CurrentAlarmSeverity := F_GetMaxSeverityRaised(Alarms := KinematicGroupAlarms, CurrentSeverity := CurrentAlarmSeverity);
END_METHOD

//! @summary Clears error flags and error IDs for this component
METHOD PUBLIC Reset : BOOL
THIS^.ResetKinGroup();
F_ClearAllEventsInClass(KinematicGroupAlarms);
_ChangeParameterSeq			  := E_ChangeParameterSeq.eChangeParameterSeq_Idle;
_KinLockTrafoParam.bExecute	  := FALSE;
_KinUnlockTrafoParam.bExecute := FALSE;
_AdsWrite.WRITE				  := FALSE;
_Error						  := FALSE;
_ErrorId					  := 0;
Reset						  := SUPER^.Reset();
END_METHOD

//! @summary This method serves as the entry point for all underlying FB logic
METHOD PUBLIC CyclicLogic

//! @description This method should be called cyclically by descendant function blocks by invoking <c>SUPER^.CyclicLogic()</c>.  Alternatively, the contents of this method could be reimplemented entirely in which case a call to this method would not be necessary.
IF NOT _InitComplete THEN
	_InitComplete := Initialize();
	RETURN;
END_IF

_KinStatus := F_KinGetChnOperationState(stKinRefIn := KinematicChannelNcToPlc);
_KinConfigGroup(stAxesList := _KinAxisIds, stKinRefIn := KinematicChannelNcToPlc);
_KinConfigGroup.bExecute := FALSE;
IF _KinConfigGroup.bError THEN
	_Error	 := TRUE;
	_ErrorId := _KinConfigGroup.nErrorId;
END_IF

_KinResetGroup(nItpChannelId := KinematicChannelNcToPlc.ChnId, stKinRefIn := KinematicChannelNcToPlc, stAxesList := _KinAxisIds);
_KinResetGroup.bExecute := FALSE;
_AdsWrite();
IF KinematicGroupAlarms[E_KinematicGroup.AdsWriteErr].bRaised THEN
	_Error	 := TRUE;
	_ErrorId := _AdsWrite.ERRID;
END_IF

_KinUnlockTrafoParam();
IF _KinUnlockTrafoParam.bError THEN
	_Error	 := TRUE;
	_ErrorId := _KinUnlockTrafoParam.nErrorId;
END_IF

_KinLockTrafoParam();
IF _KinLockTrafoParam.bError THEN
	_Error	 := TRUE;
	_ErrorId := _KinLockTrafoParam.nErrorId;
END_IF

ChangeKinematicParameter();
_KinExtendedRotationRange(oidTrafo := _OidKinTrafo);
_KinExtendedRotationRange.bExecute := FALSE;
IF _KinExtendedRotationRange.bError THEN
	_Error	 := TRUE;
	_ErrorId := _KinExtendedRotationRange.nErrorId;
END_IF

_KinPresetRotation(oidTrafo := _OidKinTrafo, stRotation := _Rotation);
_KinPresetRotation.bExecute := FALSE;
IF _KinPresetRotation.bError THEN
	_Error	 := TRUE;
	_ErrorId := _KinPresetRotation.nErrorId;
END_IF

THIS^._KinematicGroupBusy := _KinConfigGroup.bBusy OR _KinResetGroup.bBusy OR _ChangeParameterSeq <> E_ChangeParameterSeq.eChangeParameterSeq_Idle OR _KinExtendedRotationRange.bBusy OR _KinPresetRotation.bBusy;
SUPER^.CyclicLogic();
END_METHOD

METHOD ActivateExtRotationRange : BOOL
IF THIS^._KinStatus <> E_KinStatus.KinStatus_Empty THEN
	Trace('Parameter Change of Kinematic not possible - Group is active!');
	RETURN;
END_IF

IF _Busy THEN
	RETURN;
END_IF

_KinExtendedRotationRange.bExecute	:= TRUE;
_KinExtendedRotationRange.bActivate := TRUE;
ActivateExtRotationRange			:= TRUE;
END_METHOD

METHOD PUBLIC BuildKinGroup : BOOL
_KinConfigGroup.bCartesianMode := TRUE;
_KinConfigGroup.bExecute	   := TRUE;
BuildKinGroup				   := TRUE;
END_METHOD

METHOD DeactivateExtRotationRange : BOOL
IF _Busy THEN
	RETURN;
END_IF

_KinExtendedRotationRange.bExecute	:= TRUE;
_KinExtendedRotationRange.bActivate := FALSE;
DeactivateExtRotationRange			:= TRUE;
END_METHOD

METHOD PUBLIC DissolveKinGroup : BOOL
_KinConfigGroup.bCartesianMode := FALSE;
_KinConfigGroup.bExecute	   := TRUE;
DissolveKinGroup			   := TRUE;
END_METHOD

METHOD PresetRotationExtRotationRange : BOOL
VAR_INPUT
	Rotation : ARRAY[1..3] OF LREAL; // Relates to 3 rotations availabe e.g. Rx, Ry, Rz.
END_VAR
IF THIS^._KinStatus <> E_KinStatus.KinStatus_Empty THEN
	Trace('Parameter Change of Kinematic not possible - Group is active!');
	RETURN;
END_IF

IF _Busy THEN
	RETURN;
END_IF

_Rotation					   := Rotation;
_KinPresetRotation.bExecute	   := TRUE;
PresetRotationExtRotationRange := TRUE;
END_METHOD

METHOD PUBLIC ResetKinGroup : BOOL
_KinResetGroup.bExecute := TRUE;
ResetKinGroup			:= TRUE;
END_METHOD

METHOD SetKinematicParameter : BOOL
VAR_INPUT
	KinPTCID : PTCID;

	(* PTCID given is Tool PTCID, If False Parameter change is requested in main Kinematic Object*)
	isToolPTCID : BOOL;
	Length		: UDINT;
	Value		: PVOID;
END_VAR
IF THIS^._KinStatus <> E_KinStatus.KinStatus_Empty THEN
	Trace('Parameter Change of Kinematic not possible - Group is active!');
	RETURN;
END_IF

IF _Busy THEN
	RETURN;
END_IF

_AdsWrite.NETID := '';
_AdsWrite.PORT	:= AMSPORT_R0_NCSAF;
IF isToolPTCID THEN
	_AdsWrite.IDXGRP			  := _OidKinTrafoTool;
	_KinUnlockTrafoParam.oidTrafo := _OidKinTrafoTool;
	_KinLockTrafoParam.oidTrafo	  := _OidKinTrafoTool;
ELSE
	_AdsWrite.IDXGRP			  := _OidKinTrafo;
	_KinUnlockTrafoParam.oidTrafo := _OidKinTrafo;
	_KinLockTrafoParam.oidTrafo	  := _OidKinTrafo;
END_IF

_AdsWrite.IDXOFFS	  := KinPTCID;
_AdsWrite.LEN		  := Length;
_AdsWrite.SRCADDR	  := Value;
_AdsWrite.TMOUT		  := T#5S;
_ChangeParameterSeq	  := E_ChangeParameterSeq.eChangeParameterSeq_Start;
SetKinematicParameter := TRUE;
END_METHOD

{attribute 'monitoring' := 'variable'}
PROPERTY PUBLIC KinematicStatus : E_KinStatus
GET
KinematicStatus := _KinStatus;
END_GET
END_PROPERTY

{attribute 'monitoring' := 'variable'}
PROPERTY PUBLIC KinMetaInfo : REFERENCE TO U_KinMetaInfo
GET
KinMetaInfo REF= _KinMetaInfoIn;
END_GET
END_PROPERTY

PROPERTY OidKinTrafo : OTCID
GET
OidKinTrafo := _OidKinTrafo;
END_GET
SET
_OidKinTrafo := OidKinTrafo;
END_SET
END_PROPERTY

PROPERTY OidKinTrafoTool : OTCID
GET
OidKinTrafoTool := _OidKinTrafoTool;
END_GET
SET
_OidKinTrafoTool := OidKinTrafoTool;
END_SET
END_PROPERTY

METHOD PROTECTED CalcKinPosition : BOOL
VAR_INPUT
	ACS : ARRAY[1..8] OF LREAL;
END_VAR

VAR_OUTPUT
	MCS : ARRAY[1..8] OF LREAL;
END_VAR

VAR_INST
	_tempOidKinTrafo   : UDINT;
	_tempKinMetaInfoIn : U_KinMetaInfo;
	_tempAcsPosition   : ARRAY[1..8] OF LREAL;
	_tempMcsPosiiton   : ARRAY[1..8] OF LREAL;
END_VAR
CASE _KinematicPositionCalculationSeq OF
	E_KinematicPositionCalculationSeq.eKinematicPositionCalculationSeq_Start:
		// Set Input for next execution
		_tempOidKinTrafo	   := _OidKinTrafo;
		_tempKinMetaInfoIn	   := _KinMetaInfoIn;
		_tempAcsPosition	   := ACS;
		_KinCalcTrafo.bForward := TRUE;
		_KinCalcTrafo.bExecute := TRUE;
		_KinCalcMcsPosition.IN := FALSE;
		IF _KinCalcTrafo.bBusy THEN
			_KinematicPositionCalculationSeq := E_KinematicPositionCalculationSeq.eKinematicPositionCalculationSeq_Calc;
		END_IF

	E_KinematicPositionCalculationSeq.eKinematicPositionCalculationSeq_Calc:
		IF _KinCalcTrafo.bDone THEN
			_KinematicPositionCalculationSeq := E_KinematicPositionCalculationSeq.eKinematicPositionCalculationSeq_Done;
			_KinCalcTrafo.bExecute			 := FALSE;
		END_IF

		IF _KinCalcTrafo.bError THEN
			_KinematicPositionCalculationSeq := E_KinematicPositionCalculationSeq.eKinematicPositionCalculationSeq_Done; // Continue try to calculate in error case
			TRACE('Kinematic forward transformation to MCS Position failed - Check Kinematic Meta Info or mechanic configuration!');
			_KinCalcTrafo.bExecute := FALSE;
		END_IF

	E_KinematicPositionCalculationSeq.eKinematicPositionCalculationSeq_Done:
		_KinCalcMcsPosition.IN := TRUE;
		IF _KinCalcMcsPosition.Q THEN
			_KinematicPositionCalculationSeq := E_KinematicPositionCalculationSeq.eKinematicPositionCalculationSeq_Start;
		END_IF
END_CASE

_KinCalcTrafo(oidTrafo	   := _tempOidKinTrafo,
			  stAxesPosIn  := _tempAcsPosition,
			  stAxesPosOut := _tempMcsPosiiton,
			  uMetaInfoIn  := _tempKinMetaInfoIn,
			  uMetaInfoOut := _KinMetaInfoOut);

MCS := _tempMcsPosiiton;
_KinCalcMcsPosition(PT := T#250MS);
CalcKinPosition := TRUE;
END_METHOD

METHOD PRIVATE ChangeKinematicParameter : BOOL
VAR_INPUT
END_VAR
CASE _ChangeParameterSeq OF
	E_ChangeParameterSeq.eChangeParameterSeq_Idle:

	// Start set by Method SetKinematicParameter()
	E_ChangeParameterSeq.eChangeParameterSeq_Start:
		_ChangeParameterSeq := E_ChangeParameterSeq.eChangeParameterSeq_Unlock;

	E_ChangeParameterSeq.eChangeParameterSeq_Unlock:
		_KinUnlockTrafoParam.bExecute := TRUE;
		IF NOT _KinUnlockTrafoParam.bBusy AND _KinUnlockTrafoParam.bDone THEN
			_KinUnlockTrafoParam.bExecute := FALSE;
			_ChangeParameterSeq			  := E_ChangeParameterSeq.eChangeParameterSeq_Change;
		END_IF

		IF _KinUnlockTrafoParam.bError THEN
			_ChangeParameterSeq := E_ChangeParameterSeq.eChangeParameterSeq_Error;
		END_IF

	E_ChangeParameterSeq.eChangeParameterSeq_Change:
		_AdsWrite.WRITE := TRUE;
		IF _AdsWrite.BUSY THEN
			_AdsWrite.WRITE		:= FALSE;
			_ChangeParameterSeq := E_ChangeParameterSeq.eChangeParameterSeq_ChangeDone;
		END_IF

	E_ChangeParameterSeq.eChangeParameterSeq_ChangeDone:
		IF NOT _AdsWrite.BUSY AND NOT _AdsWrite.ERR THEN
			_ChangeParameterSeq := E_ChangeParameterSeq.eChangeParameterSeq_Lock;
		END_IF

		IF _AdsWrite.ERR THEN
			RaiseAlarmWithStrings(Alarm := KinematicGroupAlarms[E_KinematicGroup.AdsWriteErr], F_ADSErrorCodeExt(_AdsWrite.ERRID), '');
			_ChangeParameterSeq := E_ChangeParameterSeq.eChangeParameterSeq_Error;
		END_IF

	E_ChangeParameterSeq.eChangeParameterSeq_Lock:
		_KinLockTrafoParam.bExecute := TRUE;
		IF NOT _KinLockTrafoParam.bBusy AND _KinLockTrafoParam.bDone THEN
			_KinLockTrafoParam.bExecute := FALSE;
			_ChangeParameterSeq			:= E_ChangeParameterSeq.eChangeParameterSeq_Idle;
		END_IF

		IF _KinLockTrafoParam.bError THEN
			_ChangeParameterSeq := E_ChangeParameterSeq.eChangeParameterSeq_Error;
		END_IF

	E_ChangeParameterSeq.eChangeParameterSeq_Error:

// Error set in Monitoring
END_CASE
END_METHOD

{attribute 'monitoring' := 'variable'}
PROPERTY KinematicAxisIds : REFERENCE TO ST_KinAxes
GET
KinematicAxisIds REF= _KinAxisIds;
END_GET
END_PROPERTY

//! @summary Basic component initialization logic
METHOD PROTECTED Initialize : BOOL;

//! @description This method is called by <c>CyclicLogic()</c> as required
CASE _KinematicGroupInit OF
	E_InitializeState_KinematicGroup.eInitializeState_Start: // 
		Initialize			:= FALSE;
		_ChangeParameterSeq := E_ChangeParameterSeq.eChangeParameterSeq_Idle;
		SUPER^.Initialize();
		_KinematicGroupInit := E_InitializeState_KinematicGroup.eInitializeState_CheckLinking;

	E_InitializeState_KinematicGroup.eInitializeState_CheckLinking:
		IF F_GetMappingStatus(ADR(KinematicChannelNcToPlc), SIZEOF(KinematicChannelNcToPlc)) <> EPlcMappingStatus.MS_Mapped OR F_GetMappingStatus(ADR(KinematicChannelPlcToNc), SIZEOF(KinematicChannelPlcToNc)) <> EPlcMappingStatus.MS_Mapped THEN
			Trace(CONCAT('Programming Error init failed with Channel Links missing - ', Name));
			_Busy  := FALSE;
			_Error := TRUE;
		ELSE
			_KinematicGroupInit := E_InitializeState_KinematicGroup.eInitializeState_CheckAxisIds;
		END_IF

	E_InitializeState_KinematicGroup.eInitializeState_CheckAxisIds: //
		IF _KinAxisIds.nAxisIdsAcs[1] = 0 OR _KinAxisIds.nAxisIdsMcs[1] = 0 THEN
			Trace(CONCAT('Programming Error init failed with Axis-Ids missing - ', Name));
			_Busy  := FALSE;
			_Error := TRUE;
		ELSE
			_KinematicGroupInit := E_InitializeState_KinematicGroup.eInitializeState_CheckOid;
		END_IF

	E_InitializeState_KinematicGroup.eInitializeState_CheckOid:
		IF _OidKinTrafo = 0 THEN
			Trace(CONCAT('Programming Error init failed with Kinematic OID missing - ', Name));
			_Busy  := FALSE;
			_Error := TRUE;
		ELSE
			_KinematicGroupInit := E_InitializeState_KinematicGroup.eInitializeState_Done;
		END_IF

	E_InitializeState_KinematicGroup.eInitializeState_Done:
		_Busy	   := FALSE;
		Initialize := TRUE;
END_CASE
END_METHOD

END_FUNCTION_BLOCK

// Interfaces/I_KinematicGroup
INTERFACE I_KinematicGroup

METHOD ActivateExtRotationRange : BOOL
VAR_INPUT
END_VAR
END_METHOD

METHOD BuildKinGroup : BOOL
END_METHOD

METHOD DeactivateExtRotationRange : BOOL
VAR_INPUT
END_VAR
END_METHOD

METHOD DissolveKinGroup : BOOL
VAR_INPUT
END_VAR
END_METHOD

METHOD PresetRotationExtRotationRange : BOOL
VAR_INPUT
	Rotation : ARRAY[1..3] OF LREAL; // Relates to 3 rotations availabe e.g. Rx, Ry, Rz.
END_VAR
END_METHOD

METHOD ResetKinGroup : BOOL
VAR_INPUT
END_VAR
END_METHOD

METHOD SetKinematicParameter : BOOL
VAR_INPUT
	KinPTCID	: PTCID;
	isToolPTCID : BOOL; // PTCID given is Tool PTCID, If False Parameter change is requested in main Kinematic Object
	Length		: UDINT;
	Value		: PVOID;
END_VAR
END_METHOD

PROPERTY KinematicStatus : E_KinStatus
GET
END_GET
END_PROPERTY

PROPERTY KinMetaInfo : REFERENCE TO U_KinMetaInfo
GET
END_GET
END_PROPERTY

PROPERTY OidKinTrafo : OTCID
GET
END_GET
SET
END_SET
END_PROPERTY

PROPERTY OidKinTrafoTool : OTCID
GET
END_GET
SET
END_SET
END_PROPERTY

END_INTERFACE

// Utilities/F_ADSErrorCodeExt
(*Extended version of ADS Error Code with "Further Error codes" incl. Kinematic Error Codes*)
FUNCTION F_ADSErrorCodeExt : STRING(255)
VAR_INPUT
	ErrorId : UDINT;
END_VAR

VAR
END_VAR

CASE ErrorId OF
	// Global Error Codes 

	// 0 - 30					
	0:
		F_ADSErrorCodeExt := 'No error id found';

	1:
		F_ADSErrorCodeExt := 'Internal error.';

	2:
		F_ADSErrorCodeExt := 'No real time.';

	3:
		F_ADSErrorCodeExt := 'Allocation locked – memory error.';

	4:
		F_ADSErrorCodeExt := 'Mailbox full – the ADS message could not be sent. Reducing the number of ADS messages per cycle will help.';

	5:
		F_ADSErrorCodeExt := 'Wrong HMSG.';

	6:
		F_ADSErrorCodeExt := 'Target port not found – ADS server is not started or is not reachable.';

	7:
		F_ADSErrorCodeExt := 'Target computer not found – AMS route was not found.';

	8:
		F_ADSErrorCodeExt := 'Unknown command ID.';

	9:
		F_ADSErrorCodeExt := 'Invalid task ID.';

	10:
		F_ADSErrorCodeExt := 'No IO.';

	11:
		F_ADSErrorCodeExt := 'Unknown AMS command.';

	12:
		F_ADSErrorCodeExt := 'Win32 error.';

	13:
		F_ADSErrorCodeExt := 'Port not connected.';

	14:
		F_ADSErrorCodeExt := 'Invalid AMS length.';

	15:
		F_ADSErrorCodeExt := 'Invalid AMS Net ID.';

	16:
		F_ADSErrorCodeExt := 'Installation level is too low –TwinCAT 2 license error.';

	17:
		F_ADSErrorCodeExt := 'No debugging available.';

	18:
		F_ADSErrorCodeExt := 'Port disabled – TwinCAT system service not started.';

	19:
		F_ADSErrorCodeExt := 'Port already connected.';

	20:
		F_ADSErrorCodeExt := 'AMS Sync Win32 error.';

	21:
		F_ADSErrorCodeExt := 'AMS Sync Timeout.';

	22:
		F_ADSErrorCodeExt := 'AMS Sync error.';

	23:
		F_ADSErrorCodeExt := 'No index map for AMS Sync available.';

	24:
		F_ADSErrorCodeExt := 'Invalid AMS port.';

	25:
		F_ADSErrorCodeExt := 'No memory.';

	26:
		F_ADSErrorCodeExt := 'TCP send error.';

	27:
		F_ADSErrorCodeExt := 'Host unreachable.';

	28:
		F_ADSErrorCodeExt := 'Invalid AMS fragment.';

	29:
		F_ADSErrorCodeExt := 'TLS send error – secure ADS connection failed.';

	30:
		F_ADSErrorCodeExt := 'Access denied – secure ADS access denied.';

	// Router Error Codes 

	// 1280 - 1293					
	1280:
		F_ADSErrorCodeExt := 'Locked memory cannot be allocated.';

	1281:
		F_ADSErrorCodeExt := 'The router memory size could not be changed.';

	1282:
		F_ADSErrorCodeExt := 'The mailbox has reached the maximum number of possible messages.';

	1283:
		F_ADSErrorCodeExt := 'The Debug mailbox has reached the maximum number of possible messages.';

	1284:
		F_ADSErrorCodeExt := 'The port type is unknown.';

	1285:
		F_ADSErrorCodeExt := 'The router is not initialized.';

	1286:
		F_ADSErrorCodeExt := 'The port number is already assigned.';

	1287:
		F_ADSErrorCodeExt := 'The port is not registered.';

	1288:
		F_ADSErrorCodeExt := 'The maximum number of ports has been reached.';

	1289:
		F_ADSErrorCodeExt := 'The port is invalid.';

	1290:
		F_ADSErrorCodeExt := 'The router is not active.';

	1291:
		F_ADSErrorCodeExt := 'The mailbox has reached the maximum number for fragmented messages.';

	1292:
		F_ADSErrorCodeExt := 'A fragment timeout has occurred.';

	1293:
		F_ADSErrorCodeExt := 'The port is removed.';

	// General Error Codes 

	// 1792 - 1877							
	1792:
		F_ADSErrorCodeExt := 'General device error.';

	1793:
		F_ADSErrorCodeExt := 'Service is not supported by the server.';

	1794:
		F_ADSErrorCodeExt := 'Invalid index group.';

	1795:
		F_ADSErrorCodeExt := 'Invalid index offset.';

	1796:
		F_ADSErrorCodeExt := 'Reading or writing not permitted.';

	1797:
		F_ADSErrorCodeExt := 'Parameter size not correct.';

	1798:
		F_ADSErrorCodeExt := 'Invalid data values.';

	1799:
		F_ADSErrorCodeExt := 'Device is not ready to operate.';

	1800:
		F_ADSErrorCodeExt := 'Device is busy.';

	1801:
		F_ADSErrorCodeExt := 'Invalid operating system context. This can result from use of ADS blocks in different tasks. It may be possible to resolve this through multitasking synchronization in the PLC.';

	1802:
		F_ADSErrorCodeExt := 'Insufficient memory.';

	1803:
		F_ADSErrorCodeExt := 'Invalid parameter values.';

	1804:
		F_ADSErrorCodeExt := 'Not found (files, ...).';

	1805:
		F_ADSErrorCodeExt := 'Syntax error in file or command.';

	1806:
		F_ADSErrorCodeExt := 'Objects do not match.';

	1807:
		F_ADSErrorCodeExt := 'Object already exists.';

	1808:
		F_ADSErrorCodeExt := 'Symbol not found.';

	1809:
		F_ADSErrorCodeExt := 'Invalid symbol version. This can occur due to an online change. Create a new handle.';

	1810:
		F_ADSErrorCodeExt := 'Device (server) is in invalid state.';

	1811:
		F_ADSErrorCodeExt := 'AdsTransMode not supported.';

	1812:
		F_ADSErrorCodeExt := 'Notification handle is invalid.';

	1813:
		F_ADSErrorCodeExt := 'Notification client not registered.';

	1814:
		F_ADSErrorCodeExt := 'No further handle available.';

	1815:
		F_ADSErrorCodeExt := 'Notification size too large.';

	1816:
		F_ADSErrorCodeExt := 'Device not initialized.';

	1817:
		F_ADSErrorCodeExt := 'Device has a timeout.';

	1818:
		F_ADSErrorCodeExt := 'Interface query failed.';

	1819:
		F_ADSErrorCodeExt := 'Wrong interface requested.';

	1820:
		F_ADSErrorCodeExt := 'Class ID is invalid.';

	1821:
		F_ADSErrorCodeExt := 'Object ID is invalid.';

	1822:
		F_ADSErrorCodeExt := 'Request pending.';

	1823:
		F_ADSErrorCodeExt := 'Request is aborted.';

	1824:
		F_ADSErrorCodeExt := 'Signal warning.';

	1825:
		F_ADSErrorCodeExt := 'Invalid array index.';

	1826:
		F_ADSErrorCodeExt := 'Symbol not active.';

	1827:
		F_ADSErrorCodeExt := 'Access denied.';

	1828:
		F_ADSErrorCodeExt := 'Missing license.';

	1829:
		F_ADSErrorCodeExt := 'License expired.';

	1830:
		F_ADSErrorCodeExt := 'License exceeded.';

	1831:
		F_ADSErrorCodeExt := 'Invalid license.';

	1832:
		F_ADSErrorCodeExt := 'License problem: System ID is invalid.';

	1833:
		F_ADSErrorCodeExt := 'License not limited in time.';

	1834:
		F_ADSErrorCodeExt := 'Licensing problem: time in the future.';

	1835:
		F_ADSErrorCodeExt := 'License period too long.';

	1836:
		F_ADSErrorCodeExt := 'Exception at system startup.';

	1837:
		F_ADSErrorCodeExt := 'License file read twice.';

	1838:
		F_ADSErrorCodeExt := 'Invalid signature.';

	1839:
		F_ADSErrorCodeExt := 'Invalid certificate.';

	1840:
		F_ADSErrorCodeExt := 'Public key not known from OEM.';

	1841:
		F_ADSErrorCodeExt := 'License not valid for this system ID.';

	1842:
		F_ADSErrorCodeExt := 'Demo license prohibited.';

	1843:
		F_ADSErrorCodeExt := 'Invalid function ID.';

	1844:
		F_ADSErrorCodeExt := 'Outside the valid range.';

	1845:
		F_ADSErrorCodeExt := 'Invalid alignment.';

	1846:
		F_ADSErrorCodeExt := 'Invalid platform level.';

	1847:
		F_ADSErrorCodeExt := 'Context – forward to passive level.';

	1848:
		F_ADSErrorCodeExt := 'Context – forward to dispatch level.';

	1849:
		F_ADSErrorCodeExt := 'Context – forward to real time.';

	1856:
		F_ADSErrorCodeExt := 'Client error.';

	1857:
		F_ADSErrorCodeExt := 'Service contains an invalid parameter.';

	1858:
		F_ADSErrorCodeExt := 'Polling list is empty.';

	1859:
		F_ADSErrorCodeExt := 'Var connection already in use.';

	1860:
		F_ADSErrorCodeExt := 'The called ID is already in use.';

	1861:
		F_ADSErrorCodeExt := 'Timeout has occurred – the remote terminal is not responding in the specified ADS timeout. The route setting of the remote terminal may be configured incorrectly.';

	1862:
		F_ADSErrorCodeExt := 'Error in Win32 subsystem.';

	1863:
		F_ADSErrorCodeExt := 'Invalid client timeout value.';

	1864:
		F_ADSErrorCodeExt := 'Port not open.';

	1865:
		F_ADSErrorCodeExt := 'No AMS address.';

	1872:
		F_ADSErrorCodeExt := 'Internal error in Ads sync.';

	1873:
		F_ADSErrorCodeExt := 'Hash table overflow.';

	1874:
		F_ADSErrorCodeExt := 'Key not found in the table.';

	1875:
		F_ADSErrorCodeExt := 'No symbols in the cache.';

	1876:
		F_ADSErrorCodeExt := 'Invalid response received.';

	1877:
		F_ADSErrorCodeExt := 'Sync Port is locked.';

	// RTime Error Codes 

	// 4096 - 4122								
	4096:
		F_ADSErrorCodeExt := 'Internal error in the real-time system.';

	4097:
		F_ADSErrorCodeExt := 'Timer value is not valid.';

	4098:
		F_ADSErrorCodeExt := 'Task pointer has the invalid value 0 (zero).';

	4099:
		F_ADSErrorCodeExt := 'Stack pointer has the invalid value 0 (zero).';

	4100:
		F_ADSErrorCodeExt := 'The request task priority is already assigned.';

	4101:
		F_ADSErrorCodeExt := 'No free TCB (Task Control Block) available. The maximum number of TCBs is 64.';

	4102:
		F_ADSErrorCodeExt := 'No free semaphores available. The maximum number of semaphores is 64.';

	4103:
		F_ADSErrorCodeExt := 'No free space available in the queue. The maximum number of positions in the queue is 64.';

	4109:
		F_ADSErrorCodeExt := 'An external synchronization interrupt is already applied.';

	4110:
		F_ADSErrorCodeExt := 'No external sync interrupt applied.';

	4111:
		F_ADSErrorCodeExt := 'Application of the external synchronization interrupt has failed.';

	4112:
		F_ADSErrorCodeExt := 'Call of a service function in the wrong context';

	4119:
		F_ADSErrorCodeExt := 'Intel VT-x extension is not supported.';

	4120:
		F_ADSErrorCodeExt := 'Intel VT-x extension is not enabled in the BIOS.';

	4121:
		F_ADSErrorCodeExt := 'Missing function in Intel VT-x extension.';

	4122:
		F_ADSErrorCodeExt := 'Activation of Intel VT-x fails.';

	// TCP Winsock Error Codes 

	// 10060 - 10065									
	10060:
		F_ADSErrorCodeExt := 'A connection timeout has occurred. Error WHILE establishing the connection.';

	10061:
		F_ADSErrorCodeExt := 'Connection refused. No connection could be established because the target computer has explicitly rejected it.';

	10065:
		F_ADSErrorCodeExt := 'No route to host - a socket operation referred to an unavailable host.';

	// NC - General Error Codes 

	// 16384 - 16497
	16384:
		F_ADSErrorCodeExt := 'Internal system error in the NC on ring 0, no further details.';

	16385:
		F_ADSErrorCodeExt := 'The ring-0 memory management is not providing the required memory.';

	16386:
		F_ADSErrorCodeExt := 'Error while loading the Nc retain data.';

	16387:
		F_ADSErrorCodeExt := 'Parameter for Monitoring the NC Setpoint Issuing is Invalid.';

	16388:
		F_ADSErrorCodeExt := 'External Error.';

	16400:
		F_ADSErrorCodeExt := 'Channel identifier not allowed.';

	16401:
		F_ADSErrorCodeExt := 'Group identifier not allowed.';

	16402:
		F_ADSErrorCodeExt := 'Axis identifier not allowed.';

	16403:
		F_ADSErrorCodeExt := 'Encoder identifier not allowed.';

	16404:
		F_ADSErrorCodeExt := 'Controller identifier not allowed.';

	16405:
		F_ADSErrorCodeExt := 'Drive identifier not allowed.';

	16406:
		F_ADSErrorCodeExt := 'Table identifier not allowed.';

	16416:
		F_ADSErrorCodeExt := 'No PLC-axis interface during creation of an axis.';

	16417:
		F_ADSErrorCodeExt := 'No axis-PLC interface during creation of an axis.';

	16418:
		F_ADSErrorCodeExt := 'No encoder-I/O interface during creation of an axis.';

	16419:
		F_ADSErrorCodeExt := 'No I/O-encoder interface during creation of an axis.';

	16420:
		F_ADSErrorCodeExt := 'No drive-I/O interface during creation of an axis.';

	16421:
		F_ADSErrorCodeExt := 'No I/O-drive interface during creation of an axis.';

	16432:
		F_ADSErrorCodeExt := 'Coupling type not allowed. Unacceptable master/slave coupling type.';

	16433:
		F_ADSErrorCodeExt := 'Axis type not allowed. Unacceptable type specification during creation of an axis.';

	16434:
		F_ADSErrorCodeExt := 'Unknown Channel Type.';

	16448:
		F_ADSErrorCodeExt := 'Axis is not suitable for the intended purpose.';

	16464:
		F_ADSErrorCodeExt := 'Channel not ready for operation.';

	16465:
		F_ADSErrorCodeExt := 'Group not ready for operation.';

	16466:
		F_ADSErrorCodeExt := 'Axis not ready for operation.';

	16480:
		F_ADSErrorCodeExt := 'The channel that is to be created already exists.';

	16481:
		F_ADSErrorCodeExt := 'The group that is to be created already exists.';

	16482:
		F_ADSErrorCodeExt := 'The axis that is to be created already exists.';

	16483:
		F_ADSErrorCodeExt := 'The table that is to be created already exists, resp. it is tried internally to use an already existing table id ( e.g. for the universal flying saw).';

	16496:
		F_ADSErrorCodeExt := 'The location within the channel specified for an axis is not allowed.';

	16497:
		F_ADSErrorCodeExt := 'The location within the group specified for an axis is not allowed.';

	// NC - Channel Error Codes 

	// 16641 - 16756)					
	16641:
		F_ADSErrorCodeExt := 'Group index not allowed.';

	16642:
		F_ADSErrorCodeExt := 'The pointer to the group is invalid.';

	16643:
		F_ADSErrorCodeExt := 'No process image. It is not possible to exchange data with the PLC.';

	16644:
		F_ADSErrorCodeExt := 'Unacceptable M-function (not 0...159) detected at the execution level.';

	16645:
		F_ADSErrorCodeExt := 'No more system memory is available. This is usually the result of another error.';

	16646:
		F_ADSErrorCodeExt := 'The function is not presently available, because a similar function is already being processed.';

	16647:
		F_ADSErrorCodeExt := 'A requested function or command is not supported by the channel.';

	16648:
		F_ADSErrorCodeExt := 'Parameters to start the channel (TwinCAT-Start) are invalid.';

	16649:
		F_ADSErrorCodeExt := 'Channel function/command not executable. e.g. interpreter start is not executable because the channel is already busy, no program is loaded or in an error state.';

	16650:
		F_ADSErrorCodeExt := 'ItpGoAhead not executable. because the interpreter is not executing a decoder stop.';

	16656:
		F_ADSErrorCodeExt := 'The specified file does not exist.';

	16657:
		F_ADSErrorCodeExt := 'Syntax error during loading.';

	16658:
		F_ADSErrorCodeExt := 'Syntax error during interpretation.';

	16659:
		F_ADSErrorCodeExt := 'The NC has found a missing subroutine while loading.';

	16660:
		F_ADSErrorCodeExt := 'The capacity of the interpreter loading buffer has been exceeded.';

	16661:
		F_ADSErrorCodeExt := 'Symbolic - reserved';

	16662:
		F_ADSErrorCodeExt := 'Symbolic - reserved';

	16663:
		F_ADSErrorCodeExt := 'Subroutine incomplete. Header of subroutine is missing';

	16664:
		F_ADSErrorCodeExt := 'Error while loading the NC program. The maximum number of loadable NC programs has been reached. Possible cause: Too many sub-programs were loaded from a main program.';

	16665:
		F_ADSErrorCodeExt := 'Error while loading the NC program. The program name is too long.';

	16672:
		F_ADSErrorCodeExt := 'Divide by zero.';

	16673:
		F_ADSErrorCodeExt := 'Invalid circle parameterization. The specified circle cannot be calculated.';

	16674:
		F_ADSErrorCodeExt := 'Invalid FPU-Operation. e.g. by calculating the square root of a negative number.';

	16688:
		F_ADSErrorCodeExt := 'Stack overflow: subroutines. The NC encountered a stack overflow during execution: too many subroutine levels.';

	16689:
		F_ADSErrorCodeExt := 'Stack underflow: subroutines. The NC encountered a stack underflow during execution: too many subroutine return commands. Note: A main program must not end with a return command.';

	16690:
		F_ADSErrorCodeExt := 'Stack overflow: arithmetic unit. The NC encountered a stack overflow during execution: The calculation is too complex, or has not been correctly written.';

	16691:
		F_ADSErrorCodeExt := 'Stack underflow: arithmetic unit. The NC encountered a stack underflow during execution: The calculation is too complex, or has not been correctly written.';

	16704:
		F_ADSErrorCodeExt := 'Register index not allowed. (not R0...R999) or a pointer register contains an unacceptable value.';

	16705:
		F_ADSErrorCodeExt := 'Unacceptable G-function index. (not 0...159) during execution.';

	16706:
		F_ADSErrorCodeExt := 'Unacceptable M-function index. (not 0...159) during execution.';

	16707:
		F_ADSErrorCodeExt := 'Unacceptable extended address. (not 1...9) during execution.';

	16708:
		F_ADSErrorCodeExt := 'Unacceptable index to the internal H-function.';

	16709:
		F_ADSErrorCodeExt := 'Machine data value unacceptable. (MDB) (not 0…7).';

	16720:
		F_ADSErrorCodeExt := 'Unacceptable change of parameters for the tool compensation during execution.';

	16721:
		F_ADSErrorCodeExt := 'Cannot calculate tool compensation.';

	16722:
		F_ADSErrorCodeExt := 'Tool compensation: The plane for the tool compensation cannot be changed here. This error occurred for instance by changing the tool plane when the compensation is turned on or active.';

	16723:
		F_ADSErrorCodeExt := 'Tool compensation: The D-Word is missing or invalid by turning on the tool compensation.';

	16724:
		F_ADSErrorCodeExt := 'Tool compensation: The specified tool radius is invalid because the value is less or equal zero.';

	16725:
		F_ADSErrorCodeExt := 'Tool compensation: The tool radius cannot be changed here';

	16726:
		F_ADSErrorCodeExt := 'Tool compensation: Collision Detection Table is full.';

	16727:
		F_ADSErrorCodeExt := 'Tool compensation: Internal error while turning on the contour collision detection.';

	16728:
		F_ADSErrorCodeExt := 'Tool compensation: Internal error within the contour collision detection: update reversed geo failed.';

	16729:
		F_ADSErrorCodeExt := 'Tool compensation: Unexpected combination of geometry types by active contour collision detection.';

	16730:
		F_ADSErrorCodeExt := 'Tool compensation: Programmed inner circle is smaller than the cutter radius';

	16731:
		F_ADSErrorCodeExt := 'Tool compensation: Bottle neck detection recognized contour violation';

	16732:
		F_ADSErrorCodeExt := 'Table for corrected entries is full';

	16733:
		F_ADSErrorCodeExt := 'Input table for tangential following is full';

	16734:
		F_ADSErrorCodeExt := 'Executing table for tangential following is full';

	16735:
		F_ADSErrorCodeExt := 'Geometric entry for tangential following cannot be calculated';

	16736:
		F_ADSErrorCodeExt := 'reserved';

	16737:
		F_ADSErrorCodeExt := 'reserved';

	16738:
		F_ADSErrorCodeExt := 'The actual active interpolation rules (g-code), zero-shifts, or rotation cannot be detected';

	16752:
		F_ADSErrorCodeExt := 'The NC has found an invalid parameter while loading an NC program.';

	16753:
		F_ADSErrorCodeExt := 'Invalid contour start position.';

	16754:
		F_ADSErrorCodeExt := 'Invalid internal entry index during execution of the retrace function.';

	16755:
		F_ADSErrorCodeExt := 'Invalid default G Code. False expression/syntax in default G Code.';

	16756:
		F_ADSErrorCodeExt := 'Error while opening the default G code file.';

	// NC - Group Error Codes 

	// 16896 - 17151
	16896:
		F_ADSErrorCodeExt := 'Group ID not allowed. e.g. because it has already been assigned, is less than OR equal TO zero, OR is greater than 255. Value range: [1 ... 255]';

	16897:
		F_ADSErrorCodeExt := 'Group type not allowed.';

	16898:
		F_ADSErrorCodeExt := 'Master axis index not allowed. Value range: 0-2';

	16899:
		F_ADSErrorCodeExt := 'Slave axis index not allowed. Value range: 0-7';

	16900:
		F_ADSErrorCodeExt := 'Internal Error. Possible causes: Not enough TC router memory, internal structures and pointers are erronouos or missing, check logger';

	16901:
		F_ADSErrorCodeExt := 'Invalid cycle time for statement execution task (SAF). Value range: 0.001-0.1';

	16902:
		F_ADSErrorCodeExt := 'GROUPERR_RANGE_MAXELEMENTSINAXIS.';

	16903:
		F_ADSErrorCodeExt := 'Invalid cycle time for the statement preparation task (SVB). Value range: 0.001-1.0';

	16904:
		F_ADSErrorCodeExt := 'Single step mode not allowed.';

	16905:
		F_ADSErrorCodeExt := 'Group deactivation not allowed.';

	16906:
		F_ADSErrorCodeExt := 'Statement execution state (SAF state) not allowed. Value range: 0-5';

	16907:
		F_ADSErrorCodeExt := 'The group does not have a channel, or the channel address has not been initialized.';

	16908:
		F_ADSErrorCodeExt := 'The group does not have a master axis (or axes) or the axis address(es) has (have) not been initialized.';

	16909:
		F_ADSErrorCodeExt := 'A new master/slave coupling is to be inserted into the group, but there is no valid address for the leading master axis.';

	16910:
		F_ADSErrorCodeExt := 'A master/slave coupling is to be inserted into the group, but there is no valid address for the slave axis.';

	16911:
		F_ADSErrorCodeExt := 'A master/slave coupling is to be inserted into the group, but there is no valid address for the slave set value generator.';

	16912:
		F_ADSErrorCodeExt := 'An axis in the group does not have an encoder, or the encoder address has not been initialized.';

	16913:
		F_ADSErrorCodeExt := 'An axis in the group does not have a controller, or the controller address has not been initialized.';

	16914:
		F_ADSErrorCodeExt := 'An axis in the group does not have a drive, or the drive address has not been initialized.';

	16915:
		F_ADSErrorCodeExt := 'A group (e.g. FIFO group) does not own a master setpoint generator or a setpoint generator address has not been initialized. Possibly, there may not be enough memory available.';

	16916:
		F_ADSErrorCodeExt := 'Group/axis does not have an axis interface from the NC to the PLC, or the axis interface address has not been initialized.';

	16917:
		F_ADSErrorCodeExt := 'An existing master/slave coupling is to be removed from the group, but there is no valid address for the slave axis.';

	16918:
		F_ADSErrorCodeExt := 'Table address unknown.';

	16919:
		F_ADSErrorCodeExt := 'The NcControl address has not been initialized.';

	16920:
		F_ADSErrorCodeExt := 'Axis is blocked for commands while persistent NC data are queued.';

	16921:
		F_ADSErrorCodeExt := 'The scaling mode MASTER-AUTOOFFSET is invalid because no reference table was found.';

	16922:
		F_ADSErrorCodeExt := 'The master axis start position does not permit synchronization.';

	16923:
		F_ADSErrorCodeExt := 'Slave coupling factor (gearing factor) of 0.0 is not allowed';

	16924:
		F_ADSErrorCodeExt := 'Insertion of master axis into group not allowed';

	16925:
		F_ADSErrorCodeExt := 'Deletion of master axis from group not allowed.';

	16926:
		F_ADSErrorCodeExt := 'Function/feature is not supported from the setpoint generator.';

	16927:
		F_ADSErrorCodeExt := 'Group has not been initialized. Although the group has been created, the rest of the initialization has not been performed.';

	16928:
		F_ADSErrorCodeExt := 'Group not ready / group not ready for new task';

	16929:
		F_ADSErrorCodeExt := 'Requested set velocity is not allowed';

	16930:
		F_ADSErrorCodeExt := 'Requested target position is not allowed (master axis)';

	16931:
		F_ADSErrorCodeExt := 'No enable for controller and/or feed (Master axis).';

	16932:
		F_ADSErrorCodeExt := 'Movement smaller than one encoder increment';

	16933:
		F_ADSErrorCodeExt := 'Drive not ready during axis start';

	16934:
		F_ADSErrorCodeExt := 'Invalid parameters of the emergency stop.';

	16935:
		F_ADSErrorCodeExt := 'The setpoint generator is inactive such that no instructions are accepted.';

	16936:
		F_ADSErrorCodeExt := 'Requested traverse distance is not allowed.';

	16937:
		F_ADSErrorCodeExt := 'Requested target position is not allowed (slave axis)';

	16938:
		F_ADSErrorCodeExt := 'No enable for controller and/or feed (slave axis)';

	16939:
		F_ADSErrorCodeExt := 'The activation position (position threshold) is out of range of the actual positioning';

	16940:
		F_ADSErrorCodeExt := 'The start or activation data of the external setpoint generation are not valid';

	16941:
		F_ADSErrorCodeExt := 'For changing the dynamic parameter (accel and decel), velocity must be in constant state';

	16942:
		F_ADSErrorCodeExt := 'Jerk less than or equal to 0.0 is not allowed.';

	16943:
		F_ADSErrorCodeExt := 'Acceleration less than or equal to 0.0 is not allowed';

	16944:
		F_ADSErrorCodeExt := 'Absolute deceleration value less than or equal to 0.0 is not allowed';

	16945:
		F_ADSErrorCodeExt := 'Set velocity less than or equal to 0.0 is not allowed';

	16946:
		F_ADSErrorCodeExt := 'Loss of precision when trying a positioning.';

	16947:
		F_ADSErrorCodeExt := 'Cycle time less than or equal to 0.0 is not allowed';

	16948:
		F_ADSErrorCodeExt := 'PTP data type <intasdouble> range exceeded. Loss of precision';

	16949:
		F_ADSErrorCodeExt := 'PTP LHL velocity profile cannot be generated. (Low-High-Low)';

	16950:
		F_ADSErrorCodeExt := 'PTP HML velocity profile cannot be generated. (High-Middle-Low).';

	16951:
		F_ADSErrorCodeExt := 'Start data address is invalid.';

	16952:
		F_ADSErrorCodeExt := 'Velocity override (start override) is not allowed';

	16953:
		F_ADSErrorCodeExt := 'Start type not allowed.';

	16954:
		F_ADSErrorCodeExt := 'Velocity overflow (overshoot in the velocity). Parameterized jerk is too weak.';

	16955:
		F_ADSErrorCodeExt := 'Start parameter for the axis structure is invalid.';

	16956:
		F_ADSErrorCodeExt := 'Override generator initialization parameter invalid.';

	16957:
		F_ADSErrorCodeExt := 'Slave axis has not set value generator';

	16958:
		F_ADSErrorCodeExt := 'Table is empty. Either the SVB table or the SAF table does not contain any entries.';

	16959:
		F_ADSErrorCodeExt := 'Table is full. The SVB table or the SAF table has no more free lines.';

	16960:
		F_ADSErrorCodeExt := 'No memory available. SVB memory allocation for dynamic entry in SAF table failed.';

	16961:
		F_ADSErrorCodeExt := 'Table already contains an entry.';

	16962:
		F_ADSErrorCodeExt := 'Stop is already active.';

	16963:
		F_ADSErrorCodeExt := 'Compensation has not been carried out over the full compensation section';

	16964:
		F_ADSErrorCodeExt := 'Internal parameters for the compensation are invalid.';

	16965:
		F_ADSErrorCodeExt := 'Start of compensation refused, because compensation is already active.';

	16966:
		F_ADSErrorCodeExt := 'Stop of compensation refused, because compensation is not active.';

	16967:
		F_ADSErrorCodeExt := 'Compensation type invalid.';

	16968:
		F_ADSErrorCodeExt := 'Axis address for compensation invalid.';

	16969:
		F_ADSErrorCodeExt := 'The slave address given for on-line coupling/decoupling is invalid.';

	16970:
		F_ADSErrorCodeExt := 'Coupling velocity invalid.';

	16971:
		F_ADSErrorCodeExt := 'The velocity of what is to become the master axis and the velocity of what is to become the slave axis are not constant, so that on-line coupling is not possible.';

	16972:
		F_ADSErrorCodeExt := 'Cycle time less than or equal to 0.0 is not allowed';

	16973:
		F_ADSErrorCodeExt := 'Decoupling task not allowed.';

	16974:
		F_ADSErrorCodeExt := 'The function cannot logically be executed, e.g. some commands are not possible and not allowed for slave axes.';

	16975:
		F_ADSErrorCodeExt := 'No valid table weighting has been set.';

	16976:
		F_ADSErrorCodeExt := 'Axis type, actual position type or end position type is not allowed.';

	16977:
		F_ADSErrorCodeExt := 'Function not presently supported.';

	16978:
		F_ADSErrorCodeExt := 'State of state machine invalid.';

	16979:
		F_ADSErrorCodeExt := 'Reference cam became free too soon';

	16980:
		F_ADSErrorCodeExt := 'Clearance monitoring between activation of the hardware latch and appearance of the sync pulse';

	16981:
		F_ADSErrorCodeExt := 'No memory available. The dynamic memory allocation for the set value generator, the SVB table or the SAF table has failed.';

	16982:
		F_ADSErrorCodeExt := 'The table slave axis has no active table.';

	16983:
		F_ADSErrorCodeExt := 'Function not allowed.';

	16984:
		F_ADSErrorCodeExt := 'Stopping compensation not allowed.';

	16985:
		F_ADSErrorCodeExt := 'The slave table cannot be activated, because it is currently being used.';

	16986:
		F_ADSErrorCodeExt := 'Master or slave axis is processing a job (e.g. positioning command) while coupling is requested';

	16987:
		F_ADSErrorCodeExt := 'Slave (start) parameter is incorrect.';

	16988:
		F_ADSErrorCodeExt := 'Slave type is incorrect. The slave type does not match up to the (SVB) start type.';

	16989:
		F_ADSErrorCodeExt := 'Axis stop is already active.';

	16990:
		F_ADSErrorCodeExt := 'Maximum number of tables per slavegenerator reached.';

	16991:
		F_ADSErrorCodeExt := 'The scaling mode is invalid.';

	16992:
		F_ADSErrorCodeExt := 'Controller enable for the axis or for a coupled slave axis is not present.';

	16993:
		F_ADSErrorCodeExt := 'Table not found.';

	16994:
		F_ADSErrorCodeExt := 'Incorrect table type.';

	16995:
		F_ADSErrorCodeExt := 'Single step mode is still being processed for a group or axis and a new task was requested.';

	16996:
		F_ADSErrorCodeExt := 'Group task unknown (asynchronous table entry).';

	16997:
		F_ADSErrorCodeExt := 'Group function unknown (synchronous function)';

	16998:
		F_ADSErrorCodeExt := 'Group task for slave not allowed';

	16999:
		F_ADSErrorCodeExt := 'Group function for slave not allowed';

	17000:
		F_ADSErrorCodeExt := 'NCI Setpoint Generator is Inactive';

	17001:
		F_ADSErrorCodeExt := 'Startposition=Setpoint Position. Invalid position parameters.';

	17002:
		F_ADSErrorCodeExt := 'Parameters of the delay-generator are invalid.';

	17003:
		F_ADSErrorCodeExt := 'External parameters of the superimposed instruction are invalid.';

	17004:
		F_ADSErrorCodeExt := 'Invalid override type.';

	17005:
		F_ADSErrorCodeExt := 'Activation position under/overrun. (e.g. when exchanging a cam table).';

	17006:
		F_ADSErrorCodeExt := 'Activation impossible: Master is not moving.';

	17007:
		F_ADSErrorCodeExt := 'Activation mode not possible. Slave axis is moving.';

	17008:
		F_ADSErrorCodeExt := 'Start parameter for the compensation is invalid. Acceleration (>0) Deceleration (>0) Process velocity (>0)';

	17009:
		F_ADSErrorCodeExt := 'Start parameter for the compensation is invalid. Velocity camber is negative.';

	17010:
		F_ADSErrorCodeExt := 'Start parameter for the compensation is invalid. The section on which the compensation is to occur is not positive.';

	17011:
		F_ADSErrorCodeExt := 'Target position under/overrun.';

	17012:
		F_ADSErrorCodeExt := 'Target position will be under/overrun.';

	17013:
		F_ADSErrorCodeExt := 'Group Parameter is Invalid';

	17014:
		F_ADSErrorCodeExt := 'Joint Error at Start of Setpoint Generation';

	17015:
		F_ADSErrorCodeExt := 'Dynamic parameters not permitted.';

	17017:
		F_ADSErrorCodeExt := 'The New Target Position is Invalid or Cannot be Reached';

	17018:
		F_ADSErrorCodeExt := 'New Velocity for Moving or the Final Target Velocity is Invalid';

	17019:
		F_ADSErrorCodeExt := 'The Final Velocity or the New Target Position is Invalid';

	17020:
		F_ADSErrorCodeExt := 'The New Moving Velocity is Invalid';

	17021:
		F_ADSErrorCodeExt := 'Internal Starting Mode is Invalid';

	17022:
		F_ADSErrorCodeExt := 'A requested motion command could not be realized (BISECTION)';

	17023:
		F_ADSErrorCodeExt := 'The new target position either has been overrun or will be overrun.';

	17024:
		F_ADSErrorCodeExt := 'Group not ready / group not ready for new task';

	17025:
		F_ADSErrorCodeExt := 'The parameters of the oriented stop (O-Stop) are not admitted. The modulo-target position should not be smaller than zero and not larger or equal than the encoder mod-period.';

	17026:
		F_ADSErrorCodeExt := 'The modulo target position of the modulo-start is invalid';

	17027:
		F_ADSErrorCodeExt := 'The online change activation mode is invalid';

	17028:
		F_ADSErrorCodeExt := 'The parameterized jerk rate is smaller than the minimum jerk rate.';

	17029:
		F_ADSErrorCodeExt := 'The parameterized acceleration or deceleration is not permitted';

	17030:
		F_ADSErrorCodeExt := 'The parameterized velocity is not permitted. Less than 0';

	17031:
		F_ADSErrorCodeExt := 'A activation cannot be executed due to a pending activation';

	17032:
		F_ADSErrorCodeExt := 'Illegal combination of different cycle times within an axis group';

	17033:
		F_ADSErrorCodeExt := 'Illegal motion reversal. The previous system state is restored.';

	17034:
		F_ADSErrorCodeExt := 'Illegal moment for an axis command because there is an old axis command with activation position still active';

	17035:
		F_ADSErrorCodeExt := 'Error in the stop-calculation routine. The previous system state is restored.';

	17036:
		F_ADSErrorCodeExt := 'A command with activation position cannot fully be performed because the remaining path is too short';

	17037:
		F_ADSErrorCodeExt := 'Illegal decouple type when decoupling a slave axis.';

	17038:
		F_ADSErrorCodeExt := 'Illegal target velocity when decoupling a slave axis.';

	17039:
		F_ADSErrorCodeExt := 'The command new dynamic parameter cannot be performed since this would require a new target velocity';

	17040:
		F_ADSErrorCodeExt := 'A command with activation position cannot be performed because the axis is already in the brake phase';

	17041:
		F_ADSErrorCodeExt := 'Decouple routine of slave axis does not return a valid solution';

	17042:
		F_ADSErrorCodeExt := 'Command cannot be executed because the command buffer is full filled.';

	17043:
		F_ADSErrorCodeExt := 'Command is rejected due to an internal error in the Look Ahead.';

	17044:
		F_ADSErrorCodeExt := 'Command is rejected because the segment target velocity is not realized.';

	17045:
		F_ADSErrorCodeExt := 'Successive commands have the same final position. So the moving distance is zero.';

	17046:
		F_ADSErrorCodeExt := 'Logical positioning direction is inconsistent with the direction of the buffer command';

	17047:
		F_ADSErrorCodeExt := 'Command is rejected because the remaining positioning length is to small.';

	17050:
		F_ADSErrorCodeExt := 'Restart has Failed. There is already a motion command within the PTP buffer.';

	17051:
		F_ADSErrorCodeExt := 'Collection error for invalid start parameters. Base frequency < 0, StartFreq <1, StepCount <1 or StepCount >200, BaseAmpl <=0, StepDuration <=0, StopFreq >=1/(2*CycleTime)';

	17052:
		F_ADSErrorCodeExt := 'Reference cam is not found.';

	17053:
		F_ADSErrorCodeExt := 'Reference cam became not free';

	17054:
		F_ADSErrorCodeExt := 'IO sync pulse was not found (only when using hardware latch)';

	17055:
		F_ADSErrorCodeExt := 'The Used Buffer Mode is Unknown or not Supported in this Context';

	17056:
		F_ADSErrorCodeExt := 'Group/axis consequential error. Resulting from another causative error related to another axis within the group.';

	17057:
		F_ADSErrorCodeExt := 'Velocity reduction factor for C0/C1 transition is not allowed';

	17058:
		F_ADSErrorCodeExt := 'Critical angle at segment transition not allowed.';

	17059:
		F_ADSErrorCodeExt := 'Radius of the tolerance sphere is in an invalid range';

	17060:
		F_ADSErrorCodeExt := 'Not implemented.';

	17061:
		F_ADSErrorCodeExt := 'Start type error.';

	17062:
		F_ADSErrorCodeExt := 'Not implemented.';

	17063:
		F_ADSErrorCodeExt := 'Blending with given parameters not possible';

	17064:
		F_ADSErrorCodeExt := 'Not implemented.';

	17065:
		F_ADSErrorCodeExt := 'Curve velocity reduction method not allowed.';

	17066:
		F_ADSErrorCodeExt := 'Minimum velocity is less than 0.';

	17067:
		F_ADSErrorCodeExt := 'Power function input not allowed.';

	17068:
		F_ADSErrorCodeExt := 'Dynamic change parameter not allowed.';

	17069:
		F_ADSErrorCodeExt := 'Memory allocation error.';

	17070:
		F_ADSErrorCodeExt := 'The calculated end position differs from the end position in the nc instruction (internal error).';

	17071:
		F_ADSErrorCodeExt := 'Calculate remaining chord length is invalid.';

	17072:
		F_ADSErrorCodeExt := 'Starting the set value generator (SVB, SAF) has been refused, since the SVB task is already active.';

	17073:
		F_ADSErrorCodeExt := 'SVB parameter not allowed. Set value generator (SVB) results in logical error.';

	17074:
		F_ADSErrorCodeExt := 'Velocity reduction factor not allowed. Parameter that controls reduction of the velocity at segment transition is invalid.';

	17075:
		F_ADSErrorCodeExt := 'The helix has degenerated to a circle, and should be entered as such.';

	17076:
		F_ADSErrorCodeExt := 'The helix has degenerated to a straight line, and should be entered as such.';

	17077:
		F_ADSErrorCodeExt := 'Guider parameter not allowed.';

	17078:
		F_ADSErrorCodeExt := 'Invalid segment address. Invalid geometry or does not have a valid dynamic structure address.';

	17079:
		F_ADSErrorCodeExt := 'Unparameterized generator. The SVB generator is not yet parameterized and is therefore unable to operate.';

	17080:
		F_ADSErrorCodeExt := 'Unparameterized table. The table has no information concerning the address of the corresponding dynamic generator.';

	17082:
		F_ADSErrorCodeExt := 'The calculation of the arc length of the smoothed path failed (internal error).';

	17083:
		F_ADSErrorCodeExt := 'The radius of the tolerance ball is too small (smaller than 0.1 mm).';

	17084:
		F_ADSErrorCodeExt := 'Error while calculating DXD-Software-Limit switches (internal error)';

	17085:
		F_ADSErrorCodeExt := 'NC-Block violates software limit switches of the group. Therefore the geometric entry is denied with an error.';

	17086:
		F_ADSErrorCodeExt := 'Internal error in the evaluation of a possible software limit switch violation for the segment with the block-number xx.';

	17087:
		F_ADSErrorCodeExt := 'Invalid reference speed type.';

	17088:
		F_ADSErrorCodeExt := 'Interpolating group contains axes of an incorrect axis type. An interpolating 3D group may only contain continuously guided axes of axis type 1 (SERVO).';

	17089:
		F_ADSErrorCodeExt := 'Scalar product cannot be calculated. The length of one of the given vectors is 0.0.';

	17090:
		F_ADSErrorCodeExt := 'Inverse cosine cannot be calculated. The length of one of the given vectors is 0.0.';

	17091:
		F_ADSErrorCodeExt := 'Invalid table entry type. The given table entry type is unknown.';

	17092:
		F_ADSErrorCodeExt := 'Invalid DIN66025 information type. (INTERNAL ERROR) The given DIN66025 information type is unknown. Known types: G0, G1, G2, G3, G17, G18, G19.';

	17093:
		F_ADSErrorCodeExt := 'Invalid dimension. (INTERNAL ERROR) The CNC dimension is unknown.';

	17094:
		F_ADSErrorCodeExt := 'Geometrical object is not a straight line. The given object, interpreted as a straight line, has a length of 0.0.';

	17095:
		F_ADSErrorCodeExt := 'Geometrical object is not a circle. Interpreted as a circular arc, the given object has a length of 0.0, or an angle of 0.0 or a radius of 0.0.';

	17096:
		F_ADSErrorCodeExt := 'Geometrical object is not a helix. Interpreted as a circular arc, the given object has a length of 0.0, or an angle of 0.0, or a radius of 0.0. or a height of 0.0.';

	17097:
		F_ADSErrorCodeExt := 'Set velocity less than or equal to 0.0 is invalid.';

	17098:
		F_ADSErrorCodeExt := 'The address supplied for the look-ahead is invalid.';

	17099:
		F_ADSErrorCodeExt := 'Starting the set value generator (SAF) has been refused, since the SAF task is already active.';

	17100:
		F_ADSErrorCodeExt := 'CNC set value generation not active. Stop or change of override refused, because the set value generation is not active.';

	17101:
		F_ADSErrorCodeExt := 'CNC set value generation in the stop phase. Stop or change of override refused, because the set value generation is in the stop phase.';

	17102:
		F_ADSErrorCodeExt := 'Override not allowed. An override of less than 0.0 % or more than 100.0 % is invalid.';

	17103:
		F_ADSErrorCodeExt := 'The table address given for the initialization of the set value generator is invalid, or no valid logger connection (report file) is present.';

	17104:
		F_ADSErrorCodeExt := 'Invalid table entry type. The given table entry type is unknown.';

	17105:
		F_ADSErrorCodeExt := 'Memory allocation for the table has failed.';

	17106:
		F_ADSErrorCodeExt := 'Memory allocation for the filter has failed.';

	17107:
		F_ADSErrorCodeExt := 'Filter parameter is not allowed.';

	17108:
		F_ADSErrorCodeExt := 'Delete Distance to go (only interpolation) failed. This error occurred, if e.g. the command DelDTG was not programmed in the actual movement of the nc program.';

	17109:
		F_ADSErrorCodeExt := 'The setpoint generator of the flying saw generates incompatible values (internal error).';

	17110:
		F_ADSErrorCodeExt := 'Axis will be stopped since otherwise it will overrun its target position (old PTP setpoint generator)';

	17111:
		F_ADSErrorCodeExt := 'Internal error in the transformation from slave to master.';

	17112:
		F_ADSErrorCodeExt := 'Wrong direction in the transformation of slave to master.';

	17114:
		F_ADSErrorCodeExt := 'Parameter of Motion Function (MF) table incorrect. This may refer to the first time created data set or to online changed data.';

	17115:
		F_ADSErrorCodeExt := 'Parameter of Motion Function (MF) table incorrect. The error cause can be, that an active MF point (no IGNORE point) points at a passive MF point (IGNORE point).';

	17116:
		F_ADSErrorCodeExt := 'Internal error by using Motion Function (MF). This error cannot be solved by the user. Please ask the TwinCAT Support.';

	17117:
		F_ADSErrorCodeExt := 'Axis coupling with synchronization generator declined because of incorrect axis dynamic values';

